Yaskawa INFORM job: aprem3TRJ0.JBI

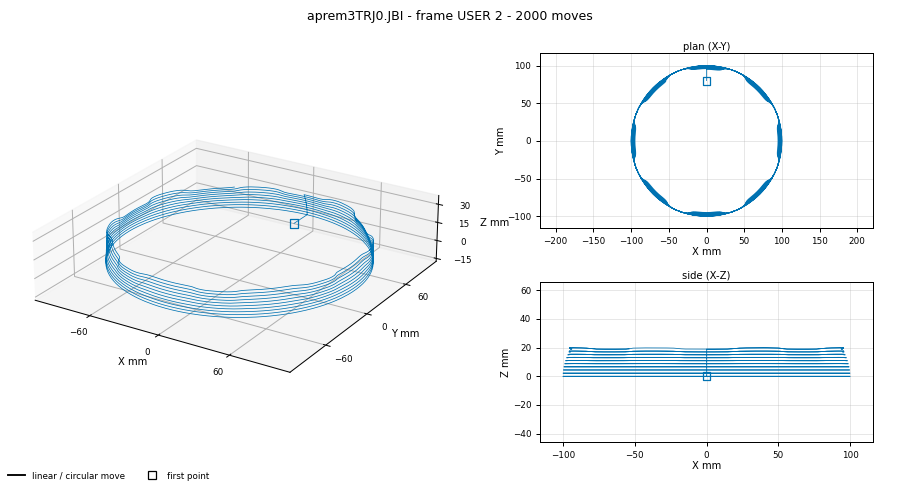
[picture p0: tool path of aprem3TRJ0.JBI in frame USER 2, 2000 of 2000 moves have a stored position in this frame; points joined in program order, loops and branches not executed]
/JOB
//NAME aprem3TRJ0
///FOLDERNAME DEMO
//POS
///NPOS 2000,0,2000,0,0,0
///USER 2
///TOOL 7
///POSTYPE USER
///RECTAN
///RCONF 1,0,0,0,0,0,0,0,0,0,0,0,0,0,0,0,0,0,0,0,0,0,0,0
C00000=0.000,80.000,0.000,-180.0000,0.0000,-0.0000
C00001=0.000,100.000,0.000,-180.0000,0.0000,-0.0000
C00002=5.792,99.832,0.000,-180.0000,-0.0000,-3.3204
C00003=10.988,99.394,0.000,-180.0000,-0.0000,-6.3084
C00004=15.564,98.781,0.000,-180.0000,-0.0000,-8.9540
C00005=18.698,98.237,0.000,-180.0000,-0.0000,-10.7765
C00006=20.854,97.801,0.000,-180.0000,-0.0000,-12.0369
C00007=22.593,97.414,0.000,-180.0000,-0.0000,-13.0576
C00008=24.351,96.990,0.000,-180.0000,-0.0000,-14.0938
C00009=26.550,96.411,0.000,-180.0000,-0.0000,-15.3967
C00010=29.248,95.627,0.000,-180.0000,-0.0000,-17.0065
C00011=32.094,94.710,0.000,-180.0000,-0.0000,-18.7198
C00012=34.739,93.772,0.000,-180.0000,-0.0000,-20.3278
C00013=37.121,92.855,0.000,-180.0000,-0.0000,-21.7902
C00014=39.410,91.907,0.000,-180.0000,-0.0000,-23.2098
C00015=41.743,90.871,0.000,-180.0000,-0.0000,-24.6724
C00016=44.276,89.664,0.000,180.0000,0.0000,-26.2801
C00017=46.937,88.300,0.000,180.0000,0.0000,-27.9935
C00018=49.400,86.946,0.000,-180.0000,-0.0000,-29.6039
C00019=51.363,85.801,0.000,-180.0000,-0.0000,-30.9060
C00020=52.906,84.858,0.000,-180.0000,-0.0000,-31.9421
C00021=54.410,83.902,0.000,-180.0000,-0.0000,-32.9632
C00022=56.242,82.685,0.000,-180.0000,-0.0000,-34.2234
C00023=58.844,80.854,0.000,-180.0000,-0.0000,-36.0464
C00024=62.512,78.053,0.000,-180.0000,-0.0000,-38.6909
C00025=66.496,74.687,0.000,-180.0000,-0.0000,-41.6796
C00026=70.711,70.711,0.000,-180.0000,-0.0000,-45.0000
C00027=74.687,66.496,0.000,-180.0000,-0.0000,-48.3204
C00028=78.053,62.512,0.000,-180.0000,-0.0000,-51.3091
C00029=80.854,58.844,0.000,180.0000,0.0000,-53.9536
C00030=82.685,56.242,0.000,-180.0000,-0.0000,-55.7766
C00031=83.902,54.410,0.000,-180.0000,-0.0000,-57.0368
C00032=84.858,52.906,0.000,-180.0000,-0.0000,-58.0579
C00033=85.801,51.363,0.000,-180.0000,-0.0000,-59.0940
C00034=86.946,49.400,0.000,-180.0000,-0.0000,-60.3961
C00035=88.300,46.937,0.000,-180.0000,-0.0000,-62.0065
C00036=89.664,44.276,0.000,-180.0000,-0.0000,-63.7199
C00037=90.871,41.743,0.000,-180.0000,-0.0000,-65.3276
C00038=91.907,39.410,0.000,-180.0000,-0.0000,-66.7902
C00039=92.855,37.121,0.000,-180.0000,-0.0000,-68.2098
C00040=93.772,34.739,0.000,-180.0000,-0.0000,-69.6722
C00041=94.710,32.094,0.000,-180.0000,-0.0000,-71.2802
C00042=95.627,29.248,0.000,-180.0000,-0.0000,-72.9935
C00043=96.411,26.550,0.000,-180.0000,-0.0000,-74.6033
C00044=96.990,24.351,0.000,-180.0000,-0.0000,-75.9062
C00045=97.414,22.593,0.000,-180.0000,-0.0000,-76.9424
C00046=97.801,20.854,0.000,-180.0000,-0.0000,-77.9631
C00047=98.237,18.698,0.000,-180.0000,-0.0000,-79.2235
C00048=98.781,15.564,0.000,-180.0000,-0.0000,-81.0460
C00049=99.394,10.988,0.000,-180.0000,-0.0000,-83.6916
C00050=99.832,5.792,0.000,-180.0000,-0.0000,-86.6796
C00051=100.000,0.000,0.000,-180.0000,-0.0000,-90.0000
C00052=99.832,-5.792,0.000,180.0000,-0.0000,-93.3204
C00053=99.394,-10.988,0.000,180.0000,-0.0000,-96.3084
C00054=98.781,-15.564,0.000,180.0000,-0.0000,-98.9540
C00055=98.237,-18.698,0.000,180.0000,-0.0000,-100.7765
C00056=97.801,-20.854,0.000,180.0000,-0.0000,-102.0369
C00057=97.414,-22.593,0.000,180.0000,-0.0000,-103.0576
C00058=96.990,-24.351,0.000,180.0000,-0.0000,-104.0938
C00059=96.411,-26.550,0.000,180.0000,-0.0000,-105.3967
C00060=95.627,-29.248,0.000,180.0000,-0.0000,-107.0065
C00061=94.710,-32.094,0.000,180.0000,-0.0000,-108.7198
C00062=93.772,-34.739,0.000,180.0000,-0.0000,-110.3278
C00063=92.855,-37.121,0.000,180.0000,-0.0000,-111.7902
C00064=91.907,-39.410,0.000,180.0000,-0.0000,-113.2098
C00065=90.871,-41.743,0.000,180.0000,-0.0000,-114.6724
C00066=89.664,-44.276,0.000,180.0000,-0.0000,-116.2801
C00067=88.300,-46.937,0.000,180.0000,-0.0000,-117.9935
C00068=86.946,-49.400,0.000,180.0000,-0.0000,-119.6039
C00069=85.801,-51.363,0.000,180.0000,-0.0000,-120.9060
C00070=84.858,-52.906,0.000,180.0000,-0.0000,-121.9421
C00071=83.902,-54.410,0.000,180.0000,-0.0000,-122.9632
C00072=82.685,-56.242,0.000,180.0000,-0.0000,-124.2234
C00073=80.854,-58.844,0.000,180.0000,-0.0000,-126.0464
C00074=78.053,-62.512,0.000,180.0000,-0.0000,-128.6909
C00075=74.687,-66.496,0.000,180.0000,-0.0000,-131.6796
C00076=70.711,-70.711,0.000,180.0000,-0.0000,-135.0000
C00077=66.496,-74.687,0.000,180.0000,-0.0000,-138.3204
C00078=62.512,-78.053,0.000,180.0000,-0.0000,-141.3091
C00079=58.844,-80.854,0.000,180.0000,-0.0000,-143.9536
C00080=56.242,-82.685,0.000,180.0000,-0.0000,-145.7766
C00081=54.410,-83.902,0.000,180.0000,-0.0000,-147.0368
C00082=52.906,-84.858,0.000,180.0000,-0.0000,-148.0579
C00083=51.363,-85.801,0.000,180.0000,-0.0000,-149.0940
C00084=49.400,-86.946,0.000,-180.0000,0.0000,-150.3961
C00085=46.937,-88.300,0.000,180.0000,-0.0000,-152.0065
C00086=44.276,-89.664,0.000,180.0000,-0.0000,-153.7199
C00087=41.743,-90.871,0.000,180.0000,-0.0000,-155.3276
C00088=39.410,-91.907,0.000,180.0000,-0.0000,-156.7902
C00089=37.121,-92.855,0.000,180.0000,-0.0000,-158.2098
C00090=34.739,-93.772,0.000,180.0000,-0.0000,-159.6722
C00091=32.094,-94.710,0.000,180.0000,-0.0000,-161.2802
C00092=29.248,-95.627,0.000,180.0000,-0.0000,-162.9935
C00093=26.550,-96.411,0.000,180.0000,-0.0000,-164.6033
C00094=24.351,-96.990,0.000,180.0000,-0.0000,-165.9062
C00095=22.593,-97.414,0.000,180.0000,-0.0000,-166.9424
C00096=20.854,-97.801,0.000,180.0000,-0.0000,-167.9631
C00097=18.698,-98.237,0.000,180.0000,-0.0000,-169.2235
C00098=15.564,-98.781,0.000,180.0000,-0.0000,-171.0460
C00099=10.988,-99.394,0.000,180.0000,-0.0000,-173.6916
C00100=5.792,-99.832,0.000,180.0000,-0.0000,-176.6796
C00101=0.000,-100.000,0.000,-180.0000,-0.0000,-180.0000
C00102=0.000,-100.000,0.000,-180.0000,-0.0000,-180.0000
C00103=-5.792,-99.832,0.000,-180.0000,-0.0000,-183.3204
C00104=-10.988,-99.394,0.000,-180.0000,-0.0000,-186.3084
C00105=-15.564,-98.781,0.000,-180.0000,-0.0000,-188.9540
C00106=-18.698,-98.237,0.000,-180.0000,-0.0000,-190.7765
C00107=-20.854,-97.801,0.000,-180.0000,-0.0000,-192.0369
C00108=-22.593,-97.414,0.000,-180.0000,-0.0000,-193.0576
C00109=-24.351,-96.990,0.000,-180.0000,-0.0000,-194.0938
C00110=-26.550,-96.411,0.000,-180.0000,-0.0000,-195.3967
C00111=-29.248,-95.627,0.000,-180.0000,-0.0000,-197.0065
C00112=-32.094,-94.710,0.000,-180.0000,-0.0000,-198.7198
C00113=-34.739,-93.772,0.000,-180.0000,-0.0000,-200.3278
C00114=-37.121,-92.855,0.000,-180.0000,-0.0000,-201.7902
C00115=-39.410,-91.907,0.000,-180.0000,-0.0000,-203.2098
C00116=-41.743,-90.871,0.000,-180.0000,-0.0000,-204.6724
C00117=-44.276,-89.664,0.000,-180.0000,-0.0000,-206.2801
C00118=-46.937,-88.300,0.000,-180.0000,-0.0000,-207.9935
C00119=-49.400,-86.946,0.000,-180.0000,-0.0000,-209.6039
C00120=-51.363,-85.801,0.000,-180.0000,-0.0000,-210.9060
C00121=-52.906,-84.858,0.000,-180.0000,-0.0000,-211.9421
C00122=-54.410,-83.902,0.000,-180.0000,-0.0000,-212.9632
C00123=-56.242,-82.685,0.000,-180.0000,-0.0000,-214.2234
C00124=-58.844,-80.854,0.000,-180.0000,-0.0000,-216.0464
C00125=-62.512,-78.053,0.000,-180.0000,-0.0000,-218.6909
C00126=-66.496,-74.687,0.000,-180.0000,-0.0000,-221.6796
C00127=-70.711,-70.711,0.000,-180.0000,-0.0000,-225.0000
C00128=-74.687,-66.496,0.000,-180.0000,-0.0000,-228.3204
C00129=-78.053,-62.512,0.000,-180.0000,-0.0000,-231.3091
C00130=-80.854,-58.844,0.000,-180.0000,-0.0000,-233.9536
C00131=-82.685,-56.242,0.000,-180.0000,-0.0000,-235.7766
C00132=-83.902,-54.410,0.000,-180.0000,-0.0000,-237.0368
C00133=-84.858,-52.906,0.000,-180.0000,-0.0000,-238.0579
C00134=-85.801,-51.363,0.000,-180.0000,-0.0000,-239.0940
C00135=-86.946,-49.400,0.000,-180.0000,-0.0000,-240.3961
C00136=-88.300,-46.937,0.000,-180.0000,-0.0000,-242.0065
C00137=-89.664,-44.276,0.000,-180.0000,-0.0000,-243.7199
C00138=-90.871,-41.743,0.000,180.0000,0.0000,-245.3276
C00139=-91.907,-39.410,0.000,180.0000,0.0000,-246.7902
C00140=-92.855,-37.121,0.000,-180.0000,-0.0000,-248.2098
C00141=-93.772,-34.739,0.000,-180.0000,-0.0000,-249.6722
C00142=-94.710,-32.094,0.000,180.0000,0.0000,-251.2802
C00143=-95.627,-29.248,0.000,180.0000,0.0000,-252.9935
C00144=-96.411,-26.550,0.000,-180.0000,-0.0000,-254.6033
C00145=-96.990,-24.351,0.000,-180.0000,-0.0000,-255.9062
C00146=-97.414,-22.593,0.000,-180.0000,-0.0000,-256.9424
C00147=-97.801,-20.854,0.000,-180.0000,-0.0000,-257.9631
C00148=-98.237,-18.698,0.000,-180.0000,-0.0000,-259.2235
C00149=-98.781,-15.564,0.000,-180.0000,-0.0000,-261.0460
C00150=-99.394,-10.988,0.000,-180.0000,-0.0000,-263.6916
C00151=-99.832,-5.792,0.000,-180.0000,-0.0000,-266.6796
C00152=-100.000,0.000,0.000,180.0000,0.0000,-270.0000
C00153=-99.832,5.792,0.000,-180.0000,0.0000,-273.3204
C00154=-99.394,10.988,0.000,-180.0000,0.0000,-276.3084
C00155=-98.781,15.564,0.000,-180.0000,0.0000,-278.9540
C00156=-98.237,18.698,0.000,-180.0000,0.0000,-280.7765
C00157=-97.801,20.854,0.000,-180.0000,0.0000,-282.0369
C00158=-97.414,22.593,0.000,-180.0000,0.0000,-283.0576
C00159=-96.990,24.351,0.000,-180.0000,0.0000,-284.0938
C00160=-96.411,26.550,0.000,-180.0000,0.0000,-285.3967
C00161=-95.627,29.248,0.000,-180.0000,0.0000,-287.0065
C00162=-94.710,32.094,0.000,-180.0000,0.0000,-288.7198
C00163=-93.772,34.739,0.000,-180.0000,0.0000,-290.3278
C00164=-92.855,37.121,0.000,-180.0000,0.0000,-291.7902
C00165=-91.907,39.410,0.000,-180.0000,0.0000,-293.2098
C00166=-90.871,41.743,0.000,-180.0000,0.0000,-294.6724
C00167=-89.664,44.276,0.000,-180.0000,0.0000,-296.2801
C00168=-88.300,46.937,0.000,-180.0000,0.0000,-297.9935
C00169=-86.946,49.400,0.000,-180.0000,0.0000,-299.6039
C00170=-85.801,51.363,0.000,-180.0000,0.0000,-300.9060
C00171=-84.858,52.906,0.000,-180.0000,0.0000,-301.9421
C00172=-83.902,54.410,0.000,-180.0000,0.0000,-302.9632
C00173=-82.685,56.242,0.000,-180.0000,0.0000,-304.2234
C00174=-80.854,58.844,0.000,-180.0000,0.0000,-306.0464
C00175=-78.053,62.512,0.000,-180.0000,0.0000,-308.6909
C00176=-74.687,66.496,0.000,-180.0000,0.0000,-311.6796
C00177=-70.711,70.711,0.000,-180.0000,0.0000,-315.0000
C00178=-66.496,74.687,0.000,-180.0000,0.0000,-318.3204
C00179=-62.512,78.053,0.000,-180.0000,0.0000,-321.3091
C00180=-58.844,80.854,0.000,-180.0000,0.0000,-323.9536
C00181=-56.242,82.685,0.000,-180.0000,0.0000,-325.7766
C00182=-54.410,83.902,0.000,-180.0000,0.0000,-327.0368
C00183=-52.906,84.858,0.000,-180.0000,0.0000,-328.0579
C00184=-51.363,85.801,0.000,-180.0000,0.0000,-329.0940
C00185=-49.400,86.946,0.000,-180.0000,0.0000,-330.3961
C00186=-46.937,88.300,0.000,-180.0000,0.0000,-332.0065
C00187=-44.276,89.664,0.000,-180.0000,0.0000,-333.7199
C00188=-41.743,90.871,0.000,-180.0000,0.0000,-335.3276
C00189=-39.410,91.907,0.000,-180.0000,0.0000,-336.7902
C00190=-37.121,92.855,0.000,-180.0000,0.0000,-338.2098
C00191=-34.739,93.772,0.000,-180.0000,0.0000,-339.6722
C00192=-32.094,94.710,0.000,-180.0000,0.0000,-341.2802
C00193=-29.248,95.627,0.000,-180.0000,0.0000,-342.9935
C00194=-26.550,96.411,0.000,-180.0000,0.0000,-344.6033
C00195=-24.351,96.990,0.000,-180.0000,0.0000,-345.9062
C00196=-22.593,97.414,0.000,-180.0000,0.0000,-346.9424
C00197=-20.854,97.801,0.000,-180.0000,0.0000,-347.9631
C00198=-18.698,98.237,0.000,-180.0000,0.0000,-349.2235
C00199=-15.564,98.781,0.000,-180.0000,0.0000,-351.0460
C00200=-10.988,99.394,0.000,-180.0000,0.0000,-353.6916
C00201=-5.792,99.832,0.000,-180.0000,0.0000,-356.6796
C00202=0.000,100.000,0.000,-180.0000,0.0000,-360.0000
C00203=0.000,99.921,2.199,-175.9398,0.0000,-360.0000
C00204=5.785,99.754,2.199,-175.9444,-0.2364,-363.3190
C00205=10.976,99.317,2.199,-175.9703,-0.4452,-366.3064
C00206=15.549,98.707,2.199,-176.1463,-0.6026,-368.9521
C00207=18.681,98.171,2.199,-176.5600,-0.6415,-370.7740
C00208=20.835,97.748,2.199,-177.1484,-0.5884,-372.0325
C00209=22.573,97.375,2.200,-177.8314,-0.4845,-373.0515
C00210=24.330,96.965,2.200,-178.5159,-0.3619,-374.0856
C00211=26.527,96.399,2.200,-179.1045,-0.2425,-375.3858
C00212=29.226,95.625,2.200,-179.5721,-0.1295,-376.9948
C00213=32.077,94.713,2.200,-179.8787,-0.0409,-378.7100
C00214=34.728,93.776,2.200,-179.9807,-0.0071,-380.3211
C00215=37.118,92.856,2.200,-179.9977,-0.0009,-381.7884
C00216=39.413,91.905,2.200,-179.9978,-0.0010,-383.2118
C00217=41.753,90.866,2.200,-179.9813,-0.0086,-384.6788
C00218=44.291,89.654,2.200,-179.8853,-0.0569,-386.2904
C00219=46.951,88.283,2.200,-179.6059,-0.2110,-388.0051
C00220=49.407,86.922,2.200,-179.1953,-0.4618,-389.6142
C00221=51.360,85.768,2.200,-178.6947,-0.7937,-390.9142
C00222=52.893,84.816,2.200,-178.1239,-1.1914,-391.9485
C00223=54.385,83.851,2.199,-177.5673,-1.6016,-392.9671
C00224=56.208,82.627,2.199,-177.1135,-1.9809,-394.2260
C00225=58.802,80.791,2.199,-176.8480,-2.3017,-396.0482
C00226=62.466,77.989,2.199,-176.8343,-2.5377,-398.6933
C00227=66.446,74.627,2.199,-176.9631,-2.7034,-401.6811
C00228=70.655,70.655,2.199,-177.1266,-2.8734,-405.0000
C00229=74.627,66.446,2.199,-177.2966,-3.0369,-408.3189
C00230=77.989,62.466,2.199,-177.4623,-3.1657,-411.3067
C00231=80.791,58.802,2.199,-177.6983,-3.1520,-413.9518
C00232=82.627,56.208,2.199,-178.0191,-2.8865,-415.7740
C00233=83.851,54.385,2.199,-178.3984,-2.4327,-417.0329
C00234=84.816,52.893,2.200,-178.8086,-1.8761,-418.0515
C00235=85.768,51.360,2.200,-179.2063,-1.3053,-419.0858
C00236=86.922,49.407,2.200,-179.5382,-0.8047,-420.3858
C00237=88.283,46.951,2.200,-179.7890,-0.3941,-421.9949
C00238=89.654,44.291,2.200,-179.9431,-0.1147,-423.7096
C00239=90.866,41.753,2.200,-179.9914,-0.0187,-425.3212
C00240=91.905,39.413,2.200,-179.9990,-0.0022,-426.7882
C00241=92.856,37.118,2.200,-179.9991,-0.0023,-428.2116
C00242=93.776,34.728,2.200,-179.9929,-0.0193,-429.6789
C00243=94.713,32.077,2.200,-179.9591,-0.1213,-431.2900
C00244=95.625,29.226,2.200,-179.8705,-0.4279,-433.0052
C00245=96.399,26.527,2.200,-179.7575,-0.8955,-434.6142
C00246=96.965,24.330,2.200,-179.6381,-1.4841,-435.9144
C00247=97.375,22.573,2.200,-179.5155,-2.1686,-436.9485
C00248=97.748,20.835,2.199,-179.4116,-2.8516,-437.9675
C00249=98.171,18.681,2.199,-179.3585,-3.4400,-439.2260
C00250=98.707,15.549,2.199,-179.3974,-3.8537,-441.0479
C00251=99.317,10.976,2.199,-179.5548,-4.0297,-443.6936
C00252=99.754,5.785,2.199,-179.7636,-4.0556,-446.6810
C00253=99.921,0.000,2.199,180.0000,-4.0602,-450.0000
C00254=99.754,-5.785,2.199,179.7636,-4.0556,-453.3190
C00255=99.317,-10.976,2.199,179.5548,-4.0297,-456.3064
C00256=98.707,-15.549,2.199,179.3974,-3.8537,-458.9521
C00257=98.171,-18.681,2.199,179.3585,-3.4400,-460.7740
C00258=97.748,-20.835,2.199,179.4116,-2.8516,-462.0325
C00259=97.375,-22.573,2.200,179.5155,-2.1686,-463.0515
C00260=96.965,-24.330,2.200,179.6381,-1.4841,-464.0856
C00261=96.399,-26.527,2.200,179.7575,-0.8955,-465.3858
C00262=95.625,-29.226,2.200,179.8705,-0.4279,-466.9948
C00263=94.713,-32.077,2.200,179.9591,-0.1213,-468.7100
C00264=93.776,-34.728,2.200,179.9929,-0.0193,-470.3211
C00265=92.856,-37.118,2.200,179.9991,-0.0023,-471.7884
C00266=91.905,-39.413,2.200,179.9990,-0.0022,-473.2118
C00267=90.866,-41.753,2.200,179.9914,-0.0187,-474.6788
C00268=89.654,-44.291,2.200,179.9431,-0.1147,-476.2904
C00269=88.283,-46.951,2.200,179.7890,-0.3941,-478.0051
C00270=86.922,-49.407,2.200,179.5382,-0.8047,-479.6142
C00271=85.768,-51.360,2.200,179.2063,-1.3053,-480.9142
C00272=84.816,-52.893,2.200,178.8086,-1.8761,-481.9485
C00273=83.851,-54.385,2.199,178.3984,-2.4327,-482.9671
C00274=82.627,-56.208,2.199,178.0191,-2.8865,-484.2260
C00275=80.791,-58.802,2.199,177.6983,-3.1520,-486.0482
C00276=77.989,-62.466,2.199,177.4623,-3.1657,-488.6933
C00277=74.627,-66.446,2.199,177.2966,-3.0369,-491.6811
C00278=70.655,-70.655,2.199,177.1266,-2.8734,-495.0000
C00279=66.446,-74.627,2.199,176.9631,-2.7034,-498.3189
C00280=62.466,-77.989,2.199,176.8343,-2.5377,-501.3067
C00281=58.802,-80.791,2.199,176.8480,-2.3017,-503.9518
C00282=56.208,-82.627,2.199,177.1135,-1.9809,-505.7740
C00283=54.385,-83.851,2.199,177.5673,-1.6016,-507.0329
C00284=52.893,-84.816,2.200,178.1239,-1.1914,-508.0515
C00285=51.360,-85.768,2.200,178.6947,-0.7937,-509.0858
C00286=49.407,-86.922,2.200,179.1953,-0.4618,-510.3858
C00287=46.951,-88.283,2.200,179.6059,-0.2110,-511.9949
C00288=44.291,-89.654,2.200,179.8853,-0.0569,-513.7096
C00289=41.753,-90.866,2.200,179.9813,-0.0086,-515.3212
C00290=39.413,-91.905,2.200,179.9978,-0.0010,-516.7882
C00291=37.118,-92.856,2.200,179.9977,-0.0009,-518.2116
C00292=34.728,-93.776,2.200,179.9807,-0.0071,-519.6789
C00293=32.077,-94.713,2.200,179.8787,-0.0409,-521.2900
C00294=29.226,-95.625,2.200,179.5721,-0.1295,-523.0052
C00295=26.527,-96.399,2.200,179.1045,-0.2425,-524.6142
C00296=24.330,-96.965,2.200,178.5159,-0.3619,-525.9144
C00297=22.573,-97.375,2.200,177.8314,-0.4845,-526.9485
C00298=20.835,-97.748,2.199,177.1484,-0.5884,-527.9675
C00299=18.681,-98.171,2.199,176.5600,-0.6415,-529.2260
C00300=15.549,-98.707,2.199,176.1463,-0.6026,-531.0479
C00301=10.976,-99.317,2.199,175.9703,-0.4452,-533.6936
C00302=5.785,-99.754,2.199,175.9444,-0.2364,-536.6810
C00303=0.000,-99.921,2.199,175.9398,0.0000,-540.0000
C00304=0.000,-99.921,2.199,175.9398,0.0000,-540.0000
C00305=-5.785,-99.754,2.199,175.9444,0.2364,-543.3190
C00306=-10.976,-99.317,2.199,175.9703,0.4452,-546.3064
C00307=-15.549,-98.707,2.199,176.1463,0.6026,-548.9521
C00308=-18.681,-98.171,2.199,176.5600,0.6415,-550.7740
C00309=-20.835,-97.748,2.199,177.1484,0.5884,-552.0325
C00310=-22.573,-97.375,2.200,177.8314,0.4845,-553.0515
C00311=-24.330,-96.965,2.200,178.5159,0.3619,-554.0856
C00312=-26.527,-96.399,2.200,179.1045,0.2425,-555.3858
C00313=-29.226,-95.625,2.200,179.5721,0.1295,-556.9948
C00314=-32.077,-94.713,2.200,179.8787,0.0409,-558.7100
C00315=-34.728,-93.776,2.200,179.9807,0.0071,-560.3211
C00316=-37.118,-92.856,2.200,179.9977,0.0009,-561.7884
C00317=-39.413,-91.905,2.200,179.9978,0.0010,-563.2118
C00318=-41.753,-90.866,2.200,179.9813,0.0086,-564.6788
C00319=-44.291,-89.654,2.200,179.8853,0.0569,-566.2904
C00320=-46.951,-88.283,2.200,179.6059,0.2110,-568.0051
C00321=-49.407,-86.922,2.200,179.1953,0.4618,-569.6142
C00322=-51.360,-85.768,2.200,178.6947,0.7937,-570.9142
C00323=-52.893,-84.816,2.200,178.1239,1.1914,-571.9485
C00324=-54.385,-83.851,2.199,177.5673,1.6016,-572.9671
C00325=-56.208,-82.627,2.199,177.1135,1.9809,-574.2260
C00326=-58.802,-80.791,2.199,176.8480,2.3017,-576.0482
C00327=-62.466,-77.989,2.199,176.8343,2.5377,-578.6933
C00328=-66.446,-74.627,2.199,176.9631,2.7034,-581.6811
C00329=-70.655,-70.655,2.199,177.1266,2.8734,-585.0000
C00330=-74.627,-66.446,2.199,177.2966,3.0369,-588.3189
C00331=-77.989,-62.466,2.199,177.4623,3.1657,-591.3067
C00332=-80.791,-58.802,2.199,177.6983,3.1520,-593.9518
C00333=-82.627,-56.208,2.199,178.0191,2.8865,-595.7740
C00334=-83.851,-54.385,2.199,178.3984,2.4327,-597.0329
C00335=-84.816,-52.893,2.200,178.8086,1.8761,-598.0515
C00336=-85.768,-51.360,2.200,179.2063,1.3053,-599.0858
C00337=-86.922,-49.407,2.200,179.5382,0.8047,-600.3858
C00338=-88.283,-46.951,2.200,179.7890,0.3941,-601.9949
C00339=-89.654,-44.291,2.200,179.9431,0.1147,-603.7096
C00340=-90.866,-41.753,2.200,179.9914,0.0187,-605.3212
C00341=-91.905,-39.413,2.200,179.9990,0.0022,-606.7882
C00342=-92.856,-37.118,2.200,179.9991,0.0023,-608.2116
C00343=-93.776,-34.728,2.200,179.9929,0.0193,-609.6789
C00344=-94.713,-32.077,2.200,179.9591,0.1213,-611.2900
C00345=-95.625,-29.226,2.200,179.8705,0.4279,-613.0052
C00346=-96.399,-26.527,2.200,179.7575,0.8955,-614.6142
C00347=-96.965,-24.330,2.200,179.6381,1.4841,-615.9144
C00348=-97.375,-22.573,2.200,179.5155,2.1686,-616.9485
C00349=-97.748,-20.835,2.199,179.4116,2.8516,-617.9675
C00350=-98.171,-18.681,2.199,179.3585,3.4400,-619.2260
C00351=-98.707,-15.549,2.199,179.3974,3.8537,-621.0479
C00352=-99.317,-10.976,2.199,179.5548,4.0297,-623.6936
C00353=-99.754,-5.785,2.199,179.7636,4.0556,-626.6810
C00354=-99.921,0.000,2.199,-180.0000,4.0602,-630.0000
C00355=-99.754,5.785,2.199,-179.7636,4.0556,-633.3190
C00356=-99.317,10.976,2.199,-179.5548,4.0297,-636.3064
C00357=-98.707,15.549,2.199,-179.3974,3.8537,-638.9521
C00358=-98.171,18.681,2.199,-179.3585,3.4400,-640.7740
C00359=-97.748,20.835,2.199,-179.4116,2.8516,-642.0325
C00360=-97.375,22.573,2.200,-179.5155,2.1686,-643.0515
C00361=-96.965,24.330,2.200,-179.6381,1.4841,-644.0856
C00362=-96.399,26.527,2.200,-179.7575,0.8955,-645.3858
C00363=-95.625,29.226,2.200,-179.8705,0.4279,-646.9948
C00364=-94.713,32.077,2.200,-179.9591,0.1213,-648.7100
C00365=-93.776,34.728,2.200,-179.9929,0.0193,-650.3211
C00366=-92.856,37.118,2.200,-179.9991,0.0023,-651.7884
C00367=-91.905,39.413,2.200,-179.9990,0.0022,-653.2118
C00368=-90.866,41.753,2.200,-179.9914,0.0187,-654.6788
C00369=-89.654,44.291,2.200,-179.9431,0.1147,-656.2904
C00370=-88.283,46.951,2.200,-179.7890,0.3941,-658.0051
C00371=-86.922,49.407,2.200,-179.5382,0.8047,-659.6142
C00372=-85.768,51.360,2.200,-179.2063,1.3053,-660.9142
C00373=-84.816,52.893,2.200,-178.8086,1.8761,-661.9485
C00374=-83.851,54.385,2.199,-178.3984,2.4327,-662.9671
C00375=-82.627,56.208,2.199,-178.0191,2.8865,-664.2260
C00376=-80.791,58.802,2.199,-177.6983,3.1520,-666.0482
C00377=-77.989,62.466,2.199,-177.4623,3.1657,-668.6933
C00378=-74.627,66.446,2.199,-177.2966,3.0369,-671.6811
C00379=-70.655,70.655,2.199,-177.1266,2.8734,-675.0000
C00380=-66.446,74.627,2.199,-176.9631,2.7034,-678.3189
C00381=-62.466,77.989,2.199,-176.8343,2.5377,-681.3067
C00382=-58.802,80.791,2.199,-176.8480,2.3017,-683.9518
C00383=-56.208,82.627,2.199,-177.1135,1.9809,-685.7740
C00384=-54.385,83.851,2.199,-177.5673,1.6016,-687.0329
C00385=-52.893,84.816,2.200,-178.1239,1.1914,-688.0515
C00386=-51.360,85.768,2.200,-178.6947,0.7937,-689.0858
C00387=-49.407,86.922,2.200,-179.1953,0.4618,-690.3858
C00388=-46.951,88.283,2.200,-179.6059,0.2110,-691.9949
C00389=-44.291,89.654,2.200,-179.8853,0.0569,-693.7096
C00390=-41.753,90.866,2.200,-179.9813,0.0086,-695.3212
C00391=-39.413,91.905,2.200,-179.9978,0.0010,-696.7882
C00392=-37.118,92.856,2.200,-179.9977,0.0009,-698.2116
C00393=-34.728,93.776,2.200,-179.9807,0.0071,-699.6789
C00394=-32.077,94.713,2.200,-179.8787,0.0409,-701.2900
C00395=-29.226,95.625,2.200,-179.5721,0.1295,-703.0052
C00396=-26.527,96.399,2.200,-179.1045,0.2425,-704.6142
C00397=-24.330,96.965,2.200,-178.5159,0.3619,-705.9144
C00398=-22.573,97.375,2.200,-177.8314,0.4845,-706.9485
C00399=-20.835,97.748,2.199,-177.1484,0.5884,-707.9675
C00400=-18.681,98.171,2.199,-176.5600,0.6415,-709.2260
C00401=-15.549,98.707,2.199,-176.1463,0.6026,-711.0479
C00402=-10.976,99.317,2.199,-175.9703,0.4452,-713.6936
C00403=-5.785,99.754,2.199,-175.9444,0.2364,-716.6810
C00404=0.000,99.921,2.199,-175.9398,0.0000,-720.0000
C00405=0.000,99.691,4.387,-172.1026,0.0000,-720.0000
C00406=5.764,99.524,4.387,-172.1115,-0.4617,-723.3146
C00407=10.941,99.090,4.387,-172.1612,-0.8645,-726.3008
C00408=15.506,98.490,4.388,-172.4978,-1.1464,-728.9471
C00409=18.630,97.979,4.390,-173.2935,-1.1748,-730.7659
C00410=20.779,97.591,4.393,-174.4370,-1.0358,-732.0199
C00411=22.514,97.259,4.396,-175.7755,-0.8390,-733.0335
C00412=24.268,96.890,4.398,-177.1185,-0.6429,-734.0616
C00413=26.460,96.362,4.399,-178.2686,-0.4458,-735.3544
C00414=29.164,95.617,4.399,-179.1783,-0.2412,-736.9622
C00415=32.027,94.722,4.399,-179.7705,-0.0761,-738.6812
C00416=34.697,93.786,4.400,-179.9632,-0.0136,-740.3024
C00417=37.107,92.860,4.400,-179.9957,-0.0017,-741.7817
C00418=39.424,91.901,4.400,-179.9957,-0.0018,-743.2185
C00419=41.782,90.851,4.400,-179.9644,-0.0164,-744.6975
C00420=44.332,89.625,4.399,-179.7839,-0.1085,-746.3188
C00421=46.990,88.233,4.399,-179.2484,-0.4105,-748.0383
C00422=49.428,86.848,4.399,-178.4605,-0.9093,-749.6456
C00423=51.352,85.672,4.398,-177.5077,-1.5842,-750.9386
C00424=52.853,84.692,4.396,-176.4188,-2.3979,-751.9667
C00425=54.314,83.700,4.393,-175.3318,-3.2102,-752.9801
C00426=56.108,82.455,4.390,-174.4229,-3.9270,-754.2340
C00427=58.679,80.608,4.388,-173.8773,-4.5153,-756.0529
C00428=62.331,77.804,4.387,-173.8348,-4.9540,-758.6992
C00429=66.299,74.450,4.387,-174.0811,-5.2722,-761.6856
C00430=70.493,70.493,4.387,-174.3980,-5.6020,-765.0000
C00431=74.450,66.299,4.387,-174.7278,-5.9188,-768.3144
C00432=77.804,62.331,4.387,-175.0460,-6.1652,-771.3008
C00433=80.608,58.679,4.388,-175.4847,-6.1227,-773.9471
C00434=82.455,56.108,4.390,-176.0730,-5.5771,-775.7660
C00435=83.700,54.314,4.393,-176.7898,-4.6682,-777.0199
C00436=84.692,52.853,4.396,-177.6021,-3.5812,-778.0333
C00437=85.672,51.352,4.398,-178.4158,-2.4923,-779.0614
C00438=86.848,49.428,4.399,-179.0907,-1.5395,-780.3544
C00439=88.233,46.990,4.399,-179.5895,-0.7516,-781.9617
C00440=89.625,44.332,4.399,-179.8915,-0.2161,-783.6812
C00441=90.851,41.782,4.400,-179.9836,-0.0356,-785.3025
C00442=91.901,39.424,4.400,-179.9982,-0.0043,-786.7815
C00443=92.860,37.107,4.400,-179.9983,-0.0043,-788.2183
C00444=93.786,34.697,4.400,-179.9864,-0.0368,-789.6976
C00445=94.722,32.027,4.399,-179.9239,-0.2295,-791.3188
C00446=95.617,29.164,4.399,-179.7588,-0.8217,-793.0378
C00447=96.362,26.460,4.399,-179.5542,-1.7314,-794.6456
C00448=96.890,24.268,4.398,-179.3571,-2.8815,-795.9384
C00449=97.259,22.514,4.396,-179.1610,-4.2245,-796.9665
C00450=97.591,20.779,4.393,-178.9642,-5.5630,-797.9801
C00451=97.979,18.630,4.390,-178.8252,-6.7065,-799.2341
C00452=98.490,15.506,4.388,-178.8536,-7.5022,-801.0529
C00453=99.090,10.941,4.387,-179.1355,-7.8388,-803.6992
C00454=99.524,5.764,4.387,-179.5383,-7.8885,-806.6854
C00455=99.691,0.000,4.387,180.0000,-7.8974,-810.0000
C00456=99.524,-5.764,4.387,179.5383,-7.8885,-813.3146
C00457=99.090,-10.941,4.387,179.1355,-7.8388,-816.3008
C00458=98.490,-15.506,4.388,178.8536,-7.5022,-818.9471
C00459=97.979,-18.630,4.390,178.8252,-6.7065,-820.7659
C00460=97.591,-20.779,4.393,178.9642,-5.5630,-822.0199
C00461=97.259,-22.514,4.396,179.1610,-4.2245,-823.0335
C00462=96.890,-24.268,4.398,179.3571,-2.8815,-824.0616
C00463=96.362,-26.460,4.399,179.5542,-1.7314,-825.3544
C00464=95.617,-29.164,4.399,179.7588,-0.8217,-826.9622
C00465=94.722,-32.027,4.399,179.9239,-0.2295,-828.6812
C00466=93.786,-34.697,4.400,179.9864,-0.0368,-830.3024
C00467=92.860,-37.107,4.400,179.9983,-0.0043,-831.7817
C00468=91.901,-39.424,4.400,179.9982,-0.0043,-833.2185
C00469=90.851,-41.782,4.400,179.9836,-0.0356,-834.6975
C00470=89.625,-44.332,4.399,179.8915,-0.2161,-836.3188
C00471=88.233,-46.990,4.399,179.5895,-0.7516,-838.0383
C00472=86.848,-49.428,4.399,179.0907,-1.5395,-839.6456
C00473=85.672,-51.352,4.398,178.4158,-2.4923,-840.9386
C00474=84.692,-52.853,4.396,177.6021,-3.5812,-841.9667
C00475=83.700,-54.314,4.393,176.7898,-4.6682,-842.9801
C00476=82.455,-56.108,4.390,176.0730,-5.5771,-844.2340
C00477=80.608,-58.679,4.388,175.4847,-6.1227,-846.0529
C00478=77.804,-62.331,4.387,175.0460,-6.1652,-848.6992
C00479=74.450,-66.299,4.387,174.7278,-5.9189,-851.6856
C00480=70.493,-70.493,4.387,174.3980,-5.6020,-855.0000
C00481=66.299,-74.450,4.387,174.0812,-5.2722,-858.3144
C00482=62.331,-77.804,4.387,173.8348,-4.9540,-861.3008
C00483=58.679,-80.608,4.388,173.8773,-4.5153,-863.9471
C00484=56.108,-82.455,4.390,174.4229,-3.9270,-865.7660
C00485=54.314,-83.700,4.393,175.3318,-3.2102,-867.0199
C00486=52.853,-84.692,4.396,176.4188,-2.3979,-868.0333
C00487=51.352,-85.672,4.398,177.5077,-1.5842,-869.0614
C00488=49.428,-86.848,4.399,178.4605,-0.9093,-870.3544
C00489=46.990,-88.233,4.399,179.2484,-0.4105,-871.9617
C00490=44.332,-89.625,4.399,179.7839,-0.1085,-873.6812
C00491=41.782,-90.851,4.400,179.9644,-0.0164,-875.3025
C00492=39.424,-91.901,4.400,179.9957,-0.0018,-876.7815
C00493=37.107,-92.860,4.400,179.9957,-0.0017,-878.2183
C00494=34.697,-93.786,4.400,179.9632,-0.0136,-879.6976
C00495=32.027,-94.722,4.399,179.7705,-0.0761,-881.3188
C00496=29.164,-95.617,4.399,179.1783,-0.2412,-883.0378
C00497=26.460,-96.362,4.399,178.2686,-0.4458,-884.6456
C00498=24.268,-96.890,4.398,177.1185,-0.6429,-885.9384
C00499=22.514,-97.259,4.396,175.7755,-0.8390,-886.9665
C00500=20.779,-97.591,4.393,174.4370,-1.0358,-887.9801
C00501=18.630,-97.979,4.390,173.2935,-1.1748,-889.2341
C00502=15.506,-98.490,4.388,172.4978,-1.1464,-891.0529
C00503=10.941,-99.090,4.387,172.1612,-0.8645,-893.6992
C00504=5.764,-99.524,4.387,172.1115,-0.4617,-896.6854
C00505=0.000,-99.691,4.387,172.1026,0.0000,-900.0000
C00506=0.000,-99.691,4.387,172.1026,0.0000,-900.0000
C00507=-5.764,-99.524,4.387,172.1115,0.4617,-903.3146
C00508=-10.941,-99.090,4.387,172.1612,0.8645,-906.3008
C00509=-15.506,-98.490,4.388,172.4978,1.1464,-908.9471
C00510=-18.630,-97.979,4.390,173.2935,1.1748,-910.7659
C00511=-20.779,-97.591,4.393,174.4370,1.0358,-912.0199
C00512=-22.514,-97.259,4.396,175.7755,0.8390,-913.0335
C00513=-24.268,-96.890,4.398,177.1185,0.6429,-914.0616
C00514=-26.460,-96.362,4.399,178.2686,0.4458,-915.3544
C00515=-29.164,-95.617,4.399,179.1783,0.2412,-916.9622
C00516=-32.027,-94.722,4.399,179.7705,0.0761,-918.6812
C00517=-34.697,-93.786,4.400,179.9632,0.0136,-920.3024
C00518=-37.107,-92.860,4.400,179.9957,0.0017,-921.7817
C00519=-39.424,-91.901,4.400,179.9957,0.0018,-923.2185
C00520=-41.782,-90.851,4.400,179.9644,0.0164,-924.6975
C00521=-44.332,-89.625,4.399,179.7839,0.1085,-926.3188
C00522=-46.990,-88.233,4.399,179.2484,0.4105,-928.0383
C00523=-49.428,-86.848,4.399,178.4605,0.9093,-929.6456
C00524=-51.352,-85.672,4.398,177.5077,1.5842,-930.9386
C00525=-52.853,-84.692,4.396,176.4188,2.3979,-931.9667
C00526=-54.314,-83.700,4.393,175.3318,3.2102,-932.9801
C00527=-56.108,-82.455,4.390,174.4229,3.9270,-934.2340
C00528=-58.679,-80.608,4.388,173.8773,4.5153,-936.0529
C00529=-62.331,-77.804,4.387,173.8348,4.9540,-938.6992
C00530=-66.299,-74.450,4.387,174.0811,5.2722,-941.6856
C00531=-70.493,-70.493,4.387,174.3980,5.6020,-945.0000
C00532=-74.450,-66.299,4.387,174.7278,5.9188,-948.3144
C00533=-77.804,-62.331,4.387,175.0460,6.1652,-951.3008
C00534=-80.608,-58.679,4.388,175.4847,6.1227,-953.9471
C00535=-82.455,-56.108,4.390,176.0730,5.5771,-955.7660
C00536=-83.700,-54.314,4.393,176.7898,4.6682,-957.0199
C00537=-84.692,-52.853,4.396,177.6021,3.5812,-958.0333
C00538=-85.672,-51.352,4.398,178.4158,2.4923,-959.0614
C00539=-86.848,-49.428,4.399,179.0907,1.5395,-960.3544
C00540=-88.233,-46.990,4.399,179.5895,0.7516,-961.9617
C00541=-89.625,-44.332,4.399,179.8915,0.2161,-963.6812
C00542=-90.851,-41.782,4.400,179.9836,0.0356,-965.3025
C00543=-91.901,-39.424,4.400,179.9982,0.0043,-966.7815
C00544=-92.860,-37.107,4.400,179.9983,0.0043,-968.2183
C00545=-93.786,-34.697,4.400,179.9864,0.0368,-969.6976
C00546=-94.722,-32.027,4.399,179.9239,0.2295,-971.3188
C00547=-95.617,-29.164,4.399,179.7588,0.8217,-973.0378
C00548=-96.362,-26.460,4.399,179.5542,1.7314,-974.6456
C00549=-96.890,-24.268,4.398,179.3571,2.8815,-975.9384
C00550=-97.259,-22.514,4.396,179.1610,4.2245,-976.9665
C00551=-97.591,-20.779,4.393,178.9642,5.5630,-977.9801
C00552=-97.979,-18.630,4.390,178.8252,6.7065,-979.2341
C00553=-98.490,-15.506,4.388,178.8536,7.5022,-981.0529
C00554=-99.090,-10.941,4.387,179.1355,7.8388,-983.6992
C00555=-99.524,-5.764,4.387,179.5383,7.8885,-986.6854
C00556=-99.691,0.000,4.387,-180.0000,7.8974,-990.0000
C00557=-99.524,5.764,4.387,-179.5383,7.8885,-993.3146
C00558=-99.090,10.941,4.387,-179.1355,7.8388,-996.3008
C00559=-98.490,15.506,4.388,-178.8536,7.5022,-998.9471
C00560=-97.979,18.630,4.390,-178.8252,6.7065,-1000.7659
C00561=-97.591,20.779,4.393,-178.9642,5.5630,-1002.0199
C00562=-97.259,22.514,4.396,-179.1610,4.2245,-1003.0335
C00563=-96.890,24.268,4.398,-179.3571,2.8815,-1004.0616
C00564=-96.362,26.460,4.399,-179.5542,1.7314,-1005.3544
C00565=-95.617,29.164,4.399,-179.7588,0.8217,-1006.9622
C00566=-94.722,32.027,4.399,-179.9239,0.2295,-1008.6812
C00567=-93.786,34.697,4.400,-179.9864,0.0368,-1010.3024
C00568=-92.860,37.107,4.400,-179.9983,0.0043,-1011.7817
C00569=-91.901,39.424,4.400,-179.9982,0.0043,-1013.2185
C00570=-90.851,41.782,4.400,-179.9836,0.0356,-1014.6975
C00571=-89.625,44.332,4.399,-179.8915,0.2161,-1016.3188
C00572=-88.233,46.990,4.399,-179.5895,0.7516,-1018.0383
C00573=-86.848,49.428,4.399,-179.0907,1.5395,-1019.6456
C00574=-85.672,51.352,4.398,-178.4158,2.4923,-1020.9386
C00575=-84.692,52.853,4.396,-177.6021,3.5812,-1021.9667
C00576=-83.700,54.314,4.393,-176.7898,4.6682,-1022.9801
C00577=-82.455,56.108,4.390,-176.0730,5.5771,-1024.2340
C00578=-80.608,58.679,4.388,-175.4847,6.1227,-1026.0529
C00579=-77.804,62.331,4.387,-175.0460,6.1652,-1028.6992
C00580=-74.450,66.299,4.387,-174.7278,5.9189,-1031.6856
C00581=-70.493,70.493,4.387,-174.3980,5.6020,-1035.0000
C00582=-66.299,74.450,4.387,-174.0812,5.2722,-1038.3144
C00583=-62.331,77.804,4.387,-173.8348,4.9540,-1041.3008
C00584=-58.679,80.608,4.388,-173.8773,4.5153,-1043.9471
C00585=-56.108,82.455,4.390,-174.4229,3.9270,-1045.7660
C00586=-54.314,83.700,4.393,-175.3318,3.2102,-1047.0199
C00587=-52.853,84.692,4.396,-176.4188,2.3979,-1048.0333
C00588=-51.352,85.672,4.398,-177.5077,1.5842,-1049.0614
C00589=-49.428,86.848,4.399,-178.4605,0.9093,-1050.3544
C00590=-46.990,88.233,4.399,-179.2484,0.4105,-1051.9617
C00591=-44.332,89.625,4.399,-179.7839,0.1085,-1053.6812
C00592=-41.782,90.851,4.400,-179.9644,0.0164,-1055.3025
C00593=-39.424,91.901,4.400,-179.9957,0.0018,-1056.7815
C00594=-37.107,92.860,4.400,-179.9957,0.0017,-1058.2183
C00595=-34.697,93.786,4.400,-179.9632,0.0136,-1059.6976
C00596=-32.027,94.722,4.399,-179.7705,0.0761,-1061.3188
C00597=-29.164,95.617,4.399,-179.1783,0.2412,-1063.0378
C00598=-26.460,96.362,4.399,-178.2686,0.4458,-1064.6456
C00599=-24.268,96.890,4.398,-177.1185,0.6429,-1065.9384
C00600=-22.514,97.259,4.396,-175.7755,0.8390,-1066.9665
C00601=-20.779,97.591,4.393,-174.4370,1.0358,-1067.9801
C00602=-18.630,97.979,4.390,-173.2935,1.1748,-1069.2341
C00603=-15.506,98.490,4.388,-172.4978,1.1464,-1071.0529
C00604=-10.941,99.090,4.387,-172.1612,0.8645,-1073.6992
C00605=-5.764,99.524,4.387,-172.1115,0.4617,-1076.6854
C00606=0.000,99.691,4.387,-172.1026,0.0000,-1080.0000
C00607=0.000,99.321,6.555,-168.5288,0.0000,-1080.0000
C00608=5.730,99.155,6.555,-168.5414,-0.6746,-1083.3073
C00609=10.884,98.723,6.555,-168.6119,-1.2518,-1086.2913
C00610=15.437,98.140,6.558,-169.0875,-1.6029,-1088.9391
C00611=18.547,97.668,6.566,-170.2252,-1.5293,-1090.7524
C00612=20.687,97.336,6.576,-171.8906,-1.2412,-1091.9986
C00613=22.417,97.071,6.585,-173.8606,-0.9699,-1093.0036
C00614=24.167,96.770,6.592,-175.8319,-0.7885,-1094.0220
C00615=26.351,96.303,6.595,-177.5102,-0.5868,-1095.3030
C00616=29.062,95.605,6.597,-178.8311,-0.3259,-1096.9082
C00617=31.947,94.737,6.598,-179.6815,-0.1030,-1098.6350
C00618=34.646,93.803,6.599,-179.9483,-0.0190,-1100.2716
C00619=37.090,92.867,6.600,-179.9940,-0.0024,-1101.7712
C00620=39.440,91.893,6.600,-179.9940,-0.0026,-1103.2288
C00621=41.830,90.827,6.599,-179.9500,-0.0231,-1104.7282
C00622=44.399,89.579,6.598,-179.7019,-0.1524,-1106.3649
C00623=47.053,88.152,6.597,-178.9430,-0.5962,-1108.0920
C00624=49.464,86.729,6.595,-177.8245,-1.3465,-1109.6973
C00625=51.338,85.515,6.592,-176.4942,-2.3935,-1110.9780
C00626=52.788,84.491,6.585,-174.9692,-3.6670,-1111.9962
C00627=54.199,83.455,6.576,-173.3790,-4.8831,-1113.0013
C00628=55.947,82.176,6.566,-171.9912,-5.8773,-1114.2478
C00629=58.480,80.311,6.558,-171.1269,-6.6473,-1116.0610
C00630=62.112,77.504,6.555,-171.0284,-7.2364,-1118.7088
C00631=66.061,74.165,6.555,-171.3764,-7.6887,-1121.6924
C00632=70.230,70.230,6.555,-171.8342,-8.1658,-1125.0000
C00633=74.165,66.061,6.555,-172.3113,-8.6235,-1128.3076
C00634=77.504,62.112,6.555,-172.7636,-8.9716,-1131.2912
C00635=80.311,58.480,6.558,-173.3528,-8.8731,-1133.9390
C00636=82.176,55.947,6.566,-174.1227,-8.0088,-1135.7522
C00637=83.455,54.199,6.576,-175.1169,-6.6210,-1136.9987
C00638=84.491,52.788,6.585,-176.3330,-5.0308,-1138.0038
C00639=85.515,51.338,6.592,-177.6065,-3.5058,-1139.0220
C00640=86.729,49.464,6.595,-178.6535,-2.1755,-1140.3027
C00641=88.152,47.053,6.597,-179.4038,-1.0570,-1141.9080
C00642=89.579,44.399,6.598,-179.8476,-0.2981,-1143.6351
C00643=90.827,41.830,6.599,-179.9769,-0.0500,-1145.2718
C00644=91.893,39.440,6.600,-179.9974,-0.0060,-1146.7712
C00645=92.867,37.090,6.600,-179.9976,-0.0060,-1148.2288
C00646=93.803,34.646,6.599,-179.9810,-0.0517,-1149.7284
C00647=94.737,31.947,6.598,-179.8970,-0.3185,-1151.3650
C00648=95.605,29.062,6.597,-179.6741,-1.1689,-1153.0918
C00649=96.303,26.351,6.595,-179.4132,-2.4898,-1154.6970
C00650=96.770,24.167,6.592,-179.2115,-4.1681,-1155.9780
C00651=97.071,22.417,6.585,-179.0301,-6.1394,-1156.9964
C00652=97.336,20.687,6.576,-178.7588,-8.1094,-1158.0014
C00653=97.668,18.547,6.566,-178.4707,-9.7748,-1159.2476
C00654=98.140,15.437,6.558,-178.3971,-10.9125,-1161.0609
C00655=98.723,10.884,6.555,-178.7482,-11.3881,-1163.7087
C00656=99.155,5.730,6.555,-179.3254,-11.4586,-1166.6927
C00657=99.321,0.000,6.555,180.0000,-11.4712,-1170.0000
C00658=99.155,-5.730,6.555,179.3254,-11.4585,-1173.3073
C00659=98.723,-10.884,6.555,178.7482,-11.3882,-1176.2913
C00660=98.140,-15.437,6.558,178.3971,-10.9125,-1178.9391
C00661=97.668,-18.547,6.566,178.4707,-9.7748,-1180.7524
C00662=97.336,-20.687,6.576,178.7588,-8.1094,-1181.9986
C00663=97.071,-22.417,6.585,179.0301,-6.1394,-1183.0036
C00664=96.770,-24.167,6.592,179.2115,-4.1681,-1184.0220
C00665=96.303,-26.351,6.595,179.4132,-2.4898,-1185.3030
C00666=95.605,-29.062,6.597,179.6741,-1.1689,-1186.9082
C00667=94.737,-31.947,6.598,179.8970,-0.3185,-1188.6350
C00668=93.803,-34.646,6.599,179.9810,-0.0517,-1190.2716
C00669=92.867,-37.090,6.600,179.9976,-0.0060,-1191.7712
C00670=91.893,-39.440,6.600,179.9974,-0.0060,-1193.2288
C00671=90.827,-41.830,6.599,179.9769,-0.0500,-1194.7282
C00672=89.579,-44.399,6.598,179.8476,-0.2981,-1196.3649
C00673=88.152,-47.053,6.597,179.4038,-1.0570,-1198.0920
C00674=86.729,-49.464,6.595,178.6535,-2.1755,-1199.6973
C00675=85.515,-51.338,6.592,177.6065,-3.5058,-1200.9780
C00676=84.491,-52.788,6.585,176.3330,-5.0308,-1201.9962
C00677=83.455,-54.199,6.576,175.1169,-6.6210,-1203.0013
C00678=82.176,-55.947,6.566,174.1227,-8.0088,-1204.2478
C00679=80.311,-58.480,6.558,173.3527,-8.8731,-1206.0610
C00680=77.504,-62.112,6.555,172.7636,-8.9716,-1208.7088
C00681=74.165,-66.061,6.555,172.3113,-8.6236,-1211.6924
C00682=70.230,-70.230,6.555,171.8342,-8.1658,-1215.0000
C00683=66.061,-74.165,6.555,171.3765,-7.6887,-1218.3076
C00684=62.112,-77.504,6.555,171.0284,-7.2364,-1221.2912
C00685=58.480,-80.311,6.558,171.1269,-6.6472,-1223.9390
C00686=55.947,-82.176,6.566,171.9912,-5.8773,-1225.7522
C00687=54.199,-83.455,6.576,173.3790,-4.8831,-1226.9987
C00688=52.788,-84.491,6.585,174.9692,-3.6670,-1228.0038
C00689=51.338,-85.515,6.592,176.4942,-2.3935,-1229.0220
C00690=49.464,-86.729,6.595,177.8245,-1.3465,-1230.3027
C00691=47.053,-88.152,6.597,178.9430,-0.5962,-1231.9080
C00692=44.399,-89.579,6.598,179.7019,-0.1524,-1233.6351
C00693=41.830,-90.827,6.599,179.9500,-0.0231,-1235.2718
C00694=39.440,-91.893,6.600,179.9940,-0.0026,-1236.7712
C00695=37.090,-92.867,6.600,179.9940,-0.0024,-1238.2288
C00696=34.646,-93.803,6.599,179.9483,-0.0190,-1239.7284
C00697=31.947,-94.737,6.598,179.6815,-0.1030,-1241.3650
C00698=29.062,-95.605,6.597,178.8311,-0.3259,-1243.0918
C00699=26.351,-96.303,6.595,177.5102,-0.5868,-1244.6970
C00700=24.167,-96.770,6.592,175.8319,-0.7885,-1245.9780
C00701=22.417,-97.071,6.585,173.8606,-0.9699,-1246.9964
C00702=20.687,-97.336,6.576,171.8906,-1.2412,-1248.0014
C00703=18.547,-97.668,6.566,170.2252,-1.5293,-1249.2476
C00704=15.437,-98.140,6.558,169.0875,-1.6029,-1251.0609
C00705=10.884,-98.723,6.555,168.6119,-1.2518,-1253.7087
C00706=5.730,-99.155,6.555,168.5414,-0.6746,-1256.6927
C00707=0.000,-99.321,6.555,168.5288,0.0000,-1260.0000
C00708=0.000,-99.321,6.555,168.5288,0.0000,-1260.0000
C00709=-5.730,-99.155,6.555,168.5415,0.6746,-1263.3073
C00710=-10.884,-98.723,6.555,168.6118,1.2518,-1266.2913
C00711=-15.437,-98.140,6.558,169.0875,1.6029,-1268.9391
C00712=-18.547,-97.668,6.566,170.2252,1.5293,-1270.7524
C00713=-20.687,-97.336,6.576,171.8906,1.2412,-1271.9986
C00714=-22.417,-97.071,6.585,173.8606,0.9699,-1273.0036
C00715=-24.167,-96.770,6.592,175.8319,0.7885,-1274.0220
C00716=-26.351,-96.303,6.595,177.5102,0.5868,-1275.3030
C00717=-29.062,-95.605,6.597,178.8311,0.3259,-1276.9082
C00718=-31.947,-94.737,6.598,179.6815,0.1030,-1278.6350
C00719=-34.646,-93.803,6.599,179.9483,0.0190,-1280.2716
C00720=-37.090,-92.867,6.600,179.9940,0.0024,-1281.7712
C00721=-39.440,-91.893,6.600,179.9940,0.0026,-1283.2288
C00722=-41.830,-90.827,6.599,179.9500,0.0231,-1284.7282
C00723=-44.399,-89.579,6.598,179.7019,0.1524,-1286.3649
C00724=-47.053,-88.152,6.597,178.9430,0.5962,-1288.0920
C00725=-49.464,-86.729,6.595,177.8245,1.3465,-1289.6973
C00726=-51.338,-85.515,6.592,176.4942,2.3935,-1290.9780
C00727=-52.788,-84.491,6.585,174.9692,3.6670,-1291.9962
C00728=-54.199,-83.455,6.576,173.3790,4.8831,-1293.0013
C00729=-55.947,-82.176,6.566,171.9912,5.8773,-1294.2478
C00730=-58.480,-80.311,6.558,171.1269,6.6473,-1296.0610
C00731=-62.112,-77.504,6.555,171.0284,7.2364,-1298.7088
C00732=-66.061,-74.165,6.555,171.3764,7.6887,-1301.6924
C00733=-70.230,-70.230,6.555,171.8342,8.1658,-1305.0000
C00734=-74.165,-66.061,6.555,172.3113,8.6235,-1308.3076
C00735=-77.504,-62.112,6.555,172.7636,8.9716,-1311.2912
C00736=-80.311,-58.480,6.558,173.3528,8.8731,-1313.9390
C00737=-82.176,-55.947,6.566,174.1227,8.0088,-1315.7522
C00738=-83.455,-54.199,6.576,175.1169,6.6210,-1316.9987
C00739=-84.491,-52.788,6.585,176.3330,5.0308,-1318.0038
C00740=-85.515,-51.338,6.592,177.6065,3.5058,-1319.0220
C00741=-86.729,-49.464,6.595,178.6535,2.1755,-1320.3027
C00742=-88.152,-47.053,6.597,179.4038,1.0570,-1321.9080
C00743=-89.579,-44.399,6.598,179.8476,0.2981,-1323.6351
C00744=-90.827,-41.830,6.599,179.9769,0.0500,-1325.2718
C00745=-91.893,-39.440,6.600,179.9974,0.0060,-1326.7712
C00746=-92.867,-37.090,6.600,179.9976,0.0060,-1328.2288
C00747=-93.803,-34.646,6.599,179.9810,0.0517,-1329.7284
C00748=-94.737,-31.947,6.598,179.8970,0.3185,-1331.3650
C00749=-95.605,-29.062,6.597,179.6741,1.1689,-1333.0918
C00750=-96.303,-26.351,6.595,179.4132,2.4898,-1334.6970
C00751=-96.770,-24.167,6.592,179.2115,4.1681,-1335.9780
C00752=-97.071,-22.417,6.585,179.0301,6.1394,-1336.9964
C00753=-97.336,-20.687,6.576,178.7588,8.1094,-1338.0014
C00754=-97.668,-18.547,6.566,178.4707,9.7748,-1339.2476
C00755=-98.140,-15.437,6.558,178.3971,10.9125,-1341.0609
C00756=-98.723,-10.884,6.555,178.7482,11.3881,-1343.7087
C00757=-99.155,-5.730,6.555,179.3254,11.4586,-1346.6927
C00758=-99.321,0.000,6.555,-180.0000,11.4712,-1350.0000
C00759=-99.155,5.730,6.555,-179.3254,11.4585,-1353.3073
C00760=-98.723,10.884,6.555,-178.7482,11.3882,-1356.2913
C00761=-98.140,15.437,6.558,-178.3971,10.9125,-1358.9391
C00762=-97.668,18.547,6.566,-178.4707,9.7748,-1360.7524
C00763=-97.336,20.687,6.576,-178.7588,8.1094,-1361.9986
C00764=-97.071,22.417,6.585,-179.0301,6.1394,-1363.0036
C00765=-96.770,24.167,6.592,-179.2115,4.1681,-1364.0220
C00766=-96.303,26.351,6.595,-179.4132,2.4898,-1365.3030
C00767=-95.605,29.062,6.597,-179.6741,1.1689,-1366.9082
C00768=-94.737,31.947,6.598,-179.8970,0.3185,-1368.6350
C00769=-93.803,34.646,6.599,-179.9810,0.0517,-1370.2716
C00770=-92.867,37.090,6.600,-179.9976,0.0060,-1371.7712
C00771=-91.893,39.440,6.600,-179.9974,0.0060,-1373.2288
C00772=-90.827,41.830,6.599,-179.9769,0.0500,-1374.7282
C00773=-89.579,44.399,6.598,-179.8476,0.2981,-1376.3649
C00774=-88.152,47.053,6.597,-179.4038,1.0570,-1378.0920
C00775=-86.729,49.464,6.595,-178.6535,2.1755,-1379.6973
C00776=-85.515,51.338,6.592,-177.6065,3.5058,-1380.9780
C00777=-84.491,52.788,6.585,-176.3330,5.0308,-1381.9962
C00778=-83.455,54.199,6.576,-175.1169,6.6210,-1383.0013
C00779=-82.176,55.947,6.566,-174.1227,8.0088,-1384.2478
C00780=-80.311,58.480,6.558,-173.3527,8.8731,-1386.0610
C00781=-77.504,62.112,6.555,-172.7636,8.9716,-1388.7088
C00782=-74.165,66.061,6.555,-172.3113,8.6236,-1391.6924
C00783=-70.230,70.230,6.555,-171.8342,8.1658,-1395.0000
C00784=-66.061,74.165,6.555,-171.3765,7.6887,-1398.3076
C00785=-62.112,77.504,6.555,-171.0284,7.2364,-1401.2912
C00786=-58.480,80.311,6.558,-171.1269,6.6472,-1403.9390
C00787=-55.947,82.176,6.566,-171.9912,5.8773,-1405.7522
C00788=-54.199,83.455,6.576,-173.3790,4.8831,-1406.9987
C00789=-52.788,84.491,6.585,-174.9692,3.6670,-1408.0038
C00790=-51.338,85.515,6.592,-176.4942,2.3935,-1409.0220
C00791=-49.464,86.729,6.595,-177.8245,1.3465,-1410.3027
C00792=-47.053,88.152,6.597,-178.9430,0.5962,-1411.9080
C00793=-44.399,89.579,6.598,-179.7019,0.1524,-1413.6351
C00794=-41.830,90.827,6.599,-179.9500,0.0231,-1415.2718
C00795=-39.440,91.893,6.600,-179.9940,0.0026,-1416.7712
C00796=-37.090,92.867,6.600,-179.9940,0.0024,-1418.2288
C00797=-34.646,93.803,6.599,-179.9483,0.0190,-1419.7284
C00798=-31.947,94.737,6.598,-179.6815,0.1030,-1421.3650
C00799=-29.062,95.605,6.597,-178.8311,0.3259,-1423.0918
C00800=-26.351,96.303,6.595,-177.5102,0.5868,-1424.6970
C00801=-24.167,96.770,6.592,-175.8319,0.7885,-1425.9780
C00802=-22.417,97.071,6.585,-173.8606,0.9699,-1426.9964
C00803=-20.687,97.336,6.576,-171.8906,1.2412,-1428.0014
C00804=-18.547,97.668,6.566,-170.2252,1.5293,-1429.2476
C00805=-15.437,98.140,6.558,-169.0875,1.6029,-1431.0609
C00806=-10.884,98.723,6.555,-168.6118,1.2518,-1433.7087
C00807=-5.730,99.155,6.555,-168.5415,0.6746,-1436.6927
C00808=0.000,99.321,6.555,-168.5288,0.0000,-1440.0000
C00809=0.000,98.820,8.697,-165.2395,0.0000,-1440.0000
C00810=5.684,98.656,8.697,-165.2556,-0.8746,-1443.2974
C00811=10.807,98.229,8.698,-165.3433,-1.6024,-1446.2783
C00812=15.344,97.668,8.705,-165.9346,-1.9496,-1448.9284
C00813=18.436,97.247,8.723,-167.3796,-1.6454,-1450.7347
C00814=20.563,96.991,8.745,-169.5531,-1.1205,-1451.9700
C00815=22.286,96.814,8.767,-172.1394,-0.8021,-1452.9633
C00816=24.029,96.606,8.782,-174.6912,-0.7561,-1453.9678
C00817=26.202,96.222,8.789,-176.8486,-0.6486,-1455.2327
C00818=28.922,95.588,8.792,-178.5415,-0.3776,-1456.8342
C00819=31.837,94.757,8.795,-179.6165,-0.1196,-1458.5716
C00820=34.577,93.826,8.798,-179.9364,-0.0233,-1460.2300
C00821=37.066,92.876,8.800,-179.9926,-0.0029,-1461.7565
C00822=39.463,91.883,8.800,-179.9927,-0.0031,-1463.2431
C00823=41.895,90.794,8.798,-179.9386,-0.0286,-1464.7700
C00824=44.491,89.515,8.795,-179.6442,-0.1866,-1466.4284
C00825=47.140,88.042,8.792,-178.7017,-0.7645,-1468.1658
C00826=49.511,86.567,8.789,-177.3127,-1.7714,-1469.7669
C00827=51.320,85.302,8.782,-175.7087,-3.2266,-1471.0323
C00828=52.699,84.217,8.767,-173.8629,-5.0134,-1472.0364
C00829=54.043,83.124,8.745,-171.7941,-6.6477,-1473.0299
C00830=55.728,81.800,8.723,-169.8719,-7.8577,-1474.2655
C00831=58.212,79.911,8.705,-168.6223,-8.7038,-1476.0719
C00832=61.817,77.101,8.698,-168.4305,-9.3780,-1478.7215
C00833=65.741,73.780,8.697,-168.8617,-9.9428,-1481.7023
C00834=69.877,69.877,8.697,-169.4466,-10.5535,-1485.0000
C00835=73.780,65.741,8.697,-170.0572,-11.1383,-1488.2977
C00836=77.101,61.817,8.698,-170.6220,-11.5695,-1491.2785
C00837=79.911,58.212,8.705,-171.2962,-11.3776,-1493.9281
C00838=81.800,55.728,8.723,-172.1423,-10.1281,-1495.7345
C00839=83.124,54.043,8.745,-173.3523,-8.2059,-1496.9701
C00840=84.217,52.699,8.767,-174.9866,-6.1371,-1497.9636
C00841=85.302,51.320,8.782,-176.7734,-4.2913,-1498.9677
C00842=86.567,49.511,8.789,-178.2286,-2.6873,-1500.2331
C00843=88.042,47.140,8.792,-179.2355,-1.2983,-1501.8342
C00844=89.515,44.491,8.795,-179.8134,-0.3558,-1503.5716
C00845=90.794,41.895,8.798,-179.9714,-0.0614,-1505.2300
C00846=91.883,39.463,8.800,-179.9969,-0.0073,-1506.7569
C00847=92.876,37.066,8.800,-179.9971,-0.0074,-1508.2435
C00848=93.826,34.577,8.798,-179.9767,-0.0636,-1509.7700
C00849=94.757,31.837,8.795,-179.8804,-0.3835,-1511.4284
C00850=95.588,28.922,8.792,-179.6224,-1.4585,-1513.1658
C00851=96.222,26.202,8.789,-179.3514,-3.1514,-1514.7673
C00852=96.606,24.029,8.782,-179.2439,-5.3088,-1516.0322
C00853=96.814,22.286,8.767,-179.1979,-7.8606,-1517.0367
C00854=96.991,20.563,8.745,-178.8795,-10.4469,-1518.0300
C00855=97.247,18.436,8.723,-178.3546,-12.6204,-1519.2653
C00856=97.668,15.344,8.705,-178.0504,-14.0654,-1521.0716
C00857=98.229,10.807,8.698,-178.3976,-14.6567,-1523.7217
C00858=98.656,5.684,8.697,-179.1254,-14.7444,-1526.7026
C00859=98.820,0.000,8.697,180.0000,-14.7605,-1530.0000
C00860=98.656,-5.684,8.697,179.1254,-14.7444,-1533.2974
C00861=98.229,-10.807,8.698,178.3976,-14.6567,-1536.2783
C00862=97.668,-15.344,8.705,178.0504,-14.0654,-1538.9284
C00863=97.247,-18.436,8.723,178.3546,-12.6204,-1540.7347
C00864=96.991,-20.563,8.745,178.8795,-10.4469,-1541.9700
C00865=96.814,-22.286,8.767,179.1979,-7.8606,-1542.9633
C00866=96.606,-24.029,8.782,179.2439,-5.3088,-1543.9678
C00867=96.222,-26.202,8.789,179.3514,-3.1514,-1545.2327
C00868=95.588,-28.922,8.792,179.6224,-1.4585,-1546.8342
C00869=94.757,-31.837,8.795,179.8804,-0.3835,-1548.5716
C00870=93.826,-34.577,8.798,179.9767,-0.0636,-1550.2300
C00871=92.876,-37.066,8.800,179.9971,-0.0074,-1551.7565
C00872=91.883,-39.463,8.800,179.9969,-0.0073,-1553.2431
C00873=90.794,-41.895,8.798,179.9714,-0.0614,-1554.7700
C00874=89.515,-44.491,8.795,179.8134,-0.3558,-1556.4284
C00875=88.042,-47.140,8.792,179.2355,-1.2983,-1558.1658
C00876=86.567,-49.511,8.789,178.2286,-2.6873,-1559.7669
C00877=85.302,-51.320,8.782,176.7734,-4.2913,-1561.0323
C00878=84.217,-52.699,8.767,174.9866,-6.1371,-1562.0364
C00879=83.124,-54.043,8.745,173.3523,-8.2059,-1563.0299
C00880=81.800,-55.728,8.723,172.1423,-10.1281,-1564.2655
C00881=79.911,-58.212,8.705,171.2962,-11.3777,-1566.0719
C00882=77.101,-61.817,8.698,170.6220,-11.5695,-1568.7215
C00883=73.780,-65.741,8.697,170.0572,-11.1383,-1571.7023
C00884=69.877,-69.877,8.697,169.4465,-10.5534,-1575.0000
C00885=65.741,-73.780,8.697,168.8617,-9.9428,-1578.2977
C00886=61.817,-77.101,8.698,168.4305,-9.3780,-1581.2785
C00887=58.212,-79.911,8.705,168.6224,-8.7038,-1583.9281
C00888=55.728,-81.800,8.723,169.8719,-7.8577,-1585.7345
C00889=54.043,-83.124,8.745,171.7941,-6.6477,-1586.9701
C00890=52.699,-84.217,8.767,173.8629,-5.0134,-1587.9636
C00891=51.320,-85.302,8.782,175.7087,-3.2266,-1588.9677
C00892=49.511,-86.567,8.789,177.3127,-1.7714,-1590.2331
C00893=47.140,-88.042,8.792,178.7017,-0.7645,-1591.8342
C00894=44.491,-89.515,8.795,179.6442,-0.1866,-1593.5716
C00895=41.895,-90.794,8.798,179.9386,-0.0286,-1595.2300
C00896=39.463,-91.883,8.800,179.9927,-0.0031,-1596.7569
C00897=37.066,-92.876,8.800,179.9926,-0.0029,-1598.2435
C00898=34.577,-93.826,8.798,179.9364,-0.0233,-1599.7700
C00899=31.837,-94.757,8.795,179.6165,-0.1196,-1601.4284
C00900=28.922,-95.588,8.792,178.5415,-0.3776,-1603.1658
C00901=26.202,-96.222,8.789,176.8486,-0.6486,-1604.7673
C00902=24.029,-96.606,8.782,174.6912,-0.7561,-1606.0322
C00903=22.286,-96.814,8.767,172.1394,-0.8021,-1607.0367
C00904=20.563,-96.991,8.745,169.5531,-1.1205,-1608.0300
C00905=18.436,-97.247,8.723,167.3796,-1.6454,-1609.2653
C00906=15.344,-97.668,8.705,165.9346,-1.9496,-1611.0716
C00907=10.807,-98.229,8.698,165.3433,-1.6024,-1613.7217
C00908=5.684,-98.656,8.697,165.2556,-0.8746,-1616.7026
C00909=0.000,-98.820,8.697,165.2395,0.0000,-1620.0000
C00910=0.000,-98.820,8.697,165.2395,0.0000,-1620.0000
C00911=-5.684,-98.656,8.697,165.2556,0.8746,-1623.2974
C00912=-10.807,-98.229,8.698,165.3433,1.6024,-1626.2783
C00913=-15.344,-97.668,8.705,165.9346,1.9496,-1628.9284
C00914=-18.436,-97.247,8.723,167.3796,1.6454,-1630.7347
C00915=-20.563,-96.991,8.745,169.5531,1.1205,-1631.9700
C00916=-22.286,-96.814,8.767,172.1394,0.8021,-1632.9633
C00917=-24.029,-96.606,8.782,174.6912,0.7561,-1633.9678
C00918=-26.202,-96.222,8.789,176.8486,0.6486,-1635.2327
C00919=-28.922,-95.588,8.792,178.5415,0.3776,-1636.8342
C00920=-31.837,-94.757,8.795,179.6165,0.1196,-1638.5716
C00921=-34.577,-93.826,8.798,179.9364,0.0233,-1640.2300
C00922=-37.066,-92.876,8.800,179.9926,0.0029,-1641.7565
C00923=-39.463,-91.883,8.800,179.9927,0.0031,-1643.2431
C00924=-41.895,-90.794,8.798,179.9386,0.0286,-1644.7700
C00925=-44.491,-89.515,8.795,179.6442,0.1866,-1646.4284
C00926=-47.140,-88.042,8.792,178.7017,0.7645,-1648.1658
C00927=-49.511,-86.567,8.789,177.3127,1.7714,-1649.7669
C00928=-51.320,-85.302,8.782,175.7087,3.2266,-1651.0323
C00929=-52.699,-84.217,8.767,173.8629,5.0134,-1652.0364
C00930=-54.043,-83.124,8.745,171.7941,6.6477,-1653.0299
C00931=-55.728,-81.800,8.723,169.8719,7.8577,-1654.2655
C00932=-58.212,-79.911,8.705,168.6223,8.7038,-1656.0719
C00933=-61.817,-77.101,8.698,168.4305,9.3780,-1658.7215
C00934=-65.741,-73.780,8.697,168.8617,9.9428,-1661.7023
C00935=-69.877,-69.877,8.697,169.4466,10.5535,-1665.0000
C00936=-73.780,-65.741,8.697,170.0572,11.1383,-1668.2977
C00937=-77.101,-61.817,8.698,170.6220,11.5695,-1671.2785
C00938=-79.911,-58.212,8.705,171.2962,11.3776,-1673.9281
C00939=-81.800,-55.728,8.723,172.1423,10.1281,-1675.7345
C00940=-83.124,-54.043,8.745,173.3523,8.2059,-1676.9701
C00941=-84.217,-52.699,8.767,174.9866,6.1371,-1677.9636
C00942=-85.302,-51.320,8.782,176.7734,4.2913,-1678.9677
C00943=-86.567,-49.511,8.789,178.2286,2.6873,-1680.2331
C00944=-88.042,-47.140,8.792,179.2355,1.2983,-1681.8342
C00945=-89.515,-44.491,8.795,179.8134,0.3558,-1683.5716
C00946=-90.794,-41.895,8.798,179.9714,0.0614,-1685.2300
C00947=-91.883,-39.463,8.800,179.9969,0.0073,-1686.7569
C00948=-92.876,-37.066,8.800,179.9971,0.0074,-1688.2435
C00949=-93.826,-34.577,8.798,179.9767,0.0636,-1689.7700
C00950=-94.757,-31.837,8.795,179.8804,0.3835,-1691.4284
C00951=-95.588,-28.922,8.792,179.6224,1.4585,-1693.1658
C00952=-96.222,-26.202,8.789,179.3514,3.1514,-1694.7673
C00953=-96.606,-24.029,8.782,179.2439,5.3088,-1696.0322
C00954=-96.814,-22.286,8.767,179.1979,7.8606,-1697.0367
C00955=-96.991,-20.563,8.745,178.8795,10.4469,-1698.0300
C00956=-97.247,-18.436,8.723,178.3546,12.6204,-1699.2653
C00957=-97.668,-15.344,8.705,178.0504,14.0654,-1701.0716
C00958=-98.229,-10.807,8.698,178.3976,14.6567,-1703.7217
C00959=-98.656,-5.684,8.697,179.1254,14.7444,-1706.7026
C00960=-98.820,0.000,8.697,-180.0000,14.7605,-1710.0000
C00961=-98.656,5.684,8.697,-179.1254,14.7444,-1713.2974
C00962=-98.229,10.807,8.698,-178.3976,14.6567,-1716.2783
C00963=-97.668,15.344,8.705,-178.0504,14.0654,-1718.9284
C00964=-97.247,18.436,8.723,-178.3546,12.6204,-1720.7347
C00965=-96.991,20.563,8.745,-178.8795,10.4469,-1721.9700
C00966=-96.814,22.286,8.767,-179.1979,7.8606,-1722.9633
C00967=-96.606,24.029,8.782,-179.2439,5.3088,-1723.9678
C00968=-96.222,26.202,8.789,-179.3514,3.1514,-1725.2327
C00969=-95.588,28.922,8.792,-179.6224,1.4585,-1726.8342
C00970=-94.757,31.837,8.795,-179.8804,0.3835,-1728.5716
C00971=-93.826,34.577,8.798,-179.9767,0.0636,-1730.2300
C00972=-92.876,37.066,8.800,-179.9971,0.0074,-1731.7565
C00973=-91.883,39.463,8.800,-179.9969,0.0073,-1733.2431
C00974=-90.794,41.895,8.798,-179.9714,0.0614,-1734.7700
C00975=-89.515,44.491,8.795,-179.8134,0.3558,-1736.4284
C00976=-88.042,47.140,8.792,-179.2355,1.2983,-1738.1658
C00977=-86.567,49.511,8.789,-178.2286,2.6873,-1739.7669
C00978=-85.302,51.320,8.782,-176.7734,4.2913,-1741.0323
C00979=-84.217,52.699,8.767,-174.9866,6.1371,-1742.0364
C00980=-83.124,54.043,8.745,-173.3523,8.2059,-1743.0299
C00981=-81.800,55.728,8.723,-172.1423,10.1281,-1744.2655
C00982=-79.911,58.212,8.705,-171.2962,11.3777,-1746.0719
C00983=-77.101,61.817,8.698,-170.6220,11.5695,-1748.7215
C00984=-73.780,65.741,8.697,-170.0572,11.1383,-1751.7023
C00985=-69.877,69.877,8.697,-169.4465,10.5534,-1755.0000
C00986=-65.741,73.780,8.697,-168.8617,9.9428,-1758.2977
C00987=-61.817,77.101,8.698,-168.4305,9.3780,-1761.2785
C00988=-58.212,79.911,8.705,-168.6224,8.7038,-1763.9281
C00989=-55.728,81.800,8.723,-169.8719,7.8577,-1765.7345
C00990=-54.043,83.124,8.745,-171.7941,6.6477,-1766.9701
C00991=-52.699,84.217,8.767,-173.8629,5.0134,-1767.9636
C00992=-51.320,85.302,8.782,-175.7087,3.2266,-1768.9677
C00993=-49.511,86.567,8.789,-177.3127,1.7714,-1770.2331
C00994=-47.140,88.042,8.792,-178.7017,0.7645,-1771.8342
C00995=-44.491,89.515,8.795,-179.6442,0.1866,-1773.5716
C00996=-41.895,90.794,8.798,-179.9386,0.0286,-1775.2300
C00997=-39.463,91.883,8.800,-179.9927,0.0031,-1776.7569
C00998=-37.066,92.876,8.800,-179.9926,0.0029,-1778.2435
C00999=-34.577,93.826,8.798,-179.9364,0.0233,-1779.7700
C01000=-31.837,94.757,8.795,-179.6165,0.1196,-1781.4284
C01001=-28.922,95.588,8.792,-178.5415,0.3776,-1783.1658
C01002=-26.202,96.222,8.789,-176.8486,0.6486,-1784.7673
C01003=-24.029,96.606,8.782,-174.6912,0.7561,-1786.0322
C01004=-22.286,96.814,8.767,-172.1394,0.8021,-1787.0367
C01005=-20.563,96.991,8.745,-169.5531,1.1205,-1788.0300
C01006=-18.436,97.247,8.723,-167.3796,1.6454,-1789.2653
C01007=-15.344,97.668,8.705,-165.9346,1.9496,-1791.0716
C01008=-10.807,98.229,8.698,-165.3433,1.6024,-1793.7217
C01009=-5.684,98.656,8.697,-165.2556,0.8746,-1796.7026
C01010=0.000,98.820,8.697,-165.2395,0.0000,-1800.0000
C01011=0.000,98.204,10.809,-162.2405,0.0001,-1800.0000
C01012=5.628,98.041,10.809,-162.2594,-1.0613,-1803.2854
C01013=10.712,97.620,10.809,-162.3610,-1.9132,-1806.2621
C01014=15.229,97.084,10.823,-163.0467,-2.1695,-1808.9150
C01015=18.298,96.727,10.856,-164.7843,-1.4750,-1810.7121
C01016=20.409,96.562,10.898,-167.4920,-0.6133,-1811.9342
C01017=22.123,96.495,10.937,-170.6949,-0.2914,-1812.9128
C01018=23.856,96.400,10.965,-173.7465,-0.5203,-1813.8997
C01019=26.016,96.121,10.978,-176.3051,-0.6217,-1815.1448
C01020=28.748,95.567,10.985,-178.3192,-0.3939,-1816.7421
C01021=31.699,94.782,10.991,-179.5791,-0.1255,-1818.4921
C01022=34.490,93.854,10.996,-179.9278,-0.0262,-1820.1777
C01023=37.037,92.887,11.000,-179.9917,-0.0033,-1821.7387
C01024=39.492,91.870,11.000,-179.9918,-0.0035,-1823.2613
C01025=41.977,90.753,10.996,-179.9305,-0.0325,-1824.8225
C01026=44.606,89.436,10.991,-179.6137,-0.2089,-1826.5076
C01027=47.248,87.904,10.985,-178.5329,-0.9103,-1828.2578
C01028=49.571,86.364,10.978,-176.9470,-2.1756,-1829.8549
C01029=51.296,85.034,10.965,-175.2038,-4.0647,-1831.1001
C01030=52.589,83.875,10.937,-173.1881,-6.4053,-1832.0874
C01031=53.849,82.711,10.898,-170.6621,-8.4913,-1833.0661
C01032=55.458,81.334,10.856,-168.1110,-9.8772,-1834.2883
C01033=57.880,79.417,10.823,-166.3774,-10.6897,-1836.0850
C01034=61.453,76.603,10.809,-166.0469,-11.3770,-1838.7375
C01035=65.346,73.305,10.809,-166.5413,-12.0309,-1841.7146
C01036=69.440,69.440,10.809,-167.2392,-12.7609,-1845.0000
C01037=73.305,65.346,10.809,-167.9691,-13.4586,-1848.2854
C01038=76.603,61.453,10.809,-168.6230,-13.9530,-1851.2625
C01039=79.417,57.880,10.823,-169.3103,-13.6226,-1853.9150
C01040=81.334,55.458,10.856,-170.1228,-11.8890,-1855.7117
C01041=82.711,53.849,10.898,-171.5087,-9.3379,-1856.9339
C01042=83.875,52.589,10.937,-173.5947,-6.8119,-1857.9126
C01043=85.034,51.296,10.965,-175.9353,-4.7962,-1858.8999
C01044=86.364,49.571,10.978,-177.8244,-3.0530,-1860.1451
C01045=87.904,47.248,10.985,-179.0897,-1.4671,-1861.7422
C01046=89.436,44.606,10.991,-179.7911,-0.3863,-1863.4924
C01047=90.753,41.977,10.996,-179.9675,-0.0695,-1865.1775
C01048=91.870,39.492,11.000,-179.9965,-0.0082,-1866.7387
C01049=92.887,37.037,11.000,-179.9967,-0.0083,-1868.2613
C01050=93.854,34.490,10.996,-179.9738,-0.0722,-1869.8223
C01051=94.782,31.699,10.991,-179.8745,-0.4209,-1871.5079
C01052=95.567,28.748,10.985,-179.6061,-1.6808,-1873.2579
C01053=96.121,26.016,10.978,-179.3783,-3.6949,-1874.8552
C01054=96.400,23.856,10.965,-179.4797,-6.2535,-1876.1003
C01055=96.495,22.123,10.937,-179.7086,-9.3051,-1877.0872
C01056=96.562,20.409,10.898,-179.3867,-12.5080,-1878.0658
C01057=96.727,18.298,10.856,-178.5250,-15.2157,-1879.2879
C01058=97.084,15.229,10.823,-177.8305,-16.9533,-1881.0850
C01059=97.620,10.712,10.809,-178.0868,-17.6390,-1883.7379
C01060=98.041,5.628,10.809,-178.9387,-17.7406,-1886.7146
C01061=98.204,0.000,10.809,179.9999,-17.7595,-1890.0000
C01062=98.041,-5.628,10.809,178.9388,-17.7405,-1893.2854
C01063=97.620,-10.712,10.809,178.0869,-17.6390,-1896.2621
C01064=97.084,-15.229,10.823,177.8304,-16.9533,-1898.9150
C01065=96.727,-18.298,10.856,178.5250,-15.2157,-1900.7121
C01066=96.562,-20.409,10.898,179.3867,-12.5080,-1901.9342
C01067=96.495,-22.123,10.937,179.7086,-9.3051,-1902.9128
C01068=96.400,-23.856,10.965,179.4797,-6.2535,-1903.8997
C01069=96.121,-26.016,10.978,179.3783,-3.6949,-1905.1448
C01070=95.567,-28.748,10.985,179.6061,-1.6808,-1906.7421
C01071=94.782,-31.699,10.991,179.8745,-0.4209,-1908.4921
C01072=93.854,-34.490,10.996,179.9738,-0.0722,-1910.1777
C01073=92.887,-37.037,11.000,179.9967,-0.0083,-1911.7387
C01074=91.870,-39.492,11.000,179.9965,-0.0082,-1913.2613
C01075=90.753,-41.977,10.996,179.9675,-0.0695,-1914.8225
C01076=89.436,-44.606,10.991,179.7911,-0.3863,-1916.5076
C01077=87.904,-47.248,10.985,179.0897,-1.4671,-1918.2578
C01078=86.364,-49.571,10.978,177.8244,-3.0530,-1919.8549
C01079=85.034,-51.296,10.965,175.9353,-4.7962,-1921.1001
C01080=83.875,-52.589,10.937,173.5947,-6.8119,-1922.0874
C01081=82.711,-53.849,10.898,171.5087,-9.3379,-1923.0661
C01082=81.334,-55.458,10.856,170.1228,-11.8890,-1924.2883
C01083=79.417,-57.880,10.823,169.3103,-13.6226,-1926.0850
C01084=76.603,-61.453,10.809,168.6230,-13.9531,-1928.7375
C01085=73.305,-65.346,10.809,167.9691,-13.4587,-1931.7146
C01086=69.440,-69.440,10.809,167.2391,-12.7608,-1935.0000
C01087=65.346,-73.305,10.809,166.5414,-12.0309,-1938.2854
C01088=61.453,-76.603,10.809,166.0470,-11.3770,-1941.2625
C01089=57.880,-79.417,10.823,166.3774,-10.6897,-1943.9150
C01090=55.458,-81.334,10.856,168.1110,-9.8772,-1945.7117
C01091=53.849,-82.711,10.898,170.6621,-8.4913,-1946.9339
C01092=52.589,-83.875,10.937,173.1881,-6.4053,-1947.9126
C01093=51.296,-85.034,10.965,175.2038,-4.0647,-1948.8999
C01094=49.571,-86.364,10.978,176.9470,-2.1756,-1950.1451
C01095=47.248,-87.904,10.985,178.5329,-0.9103,-1951.7422
C01096=44.606,-89.436,10.991,179.6137,-0.2089,-1953.4924
C01097=41.977,-90.753,10.996,179.9305,-0.0325,-1955.1775
C01098=39.492,-91.870,11.000,179.9918,-0.0035,-1956.7387
C01099=37.037,-92.887,11.000,179.9917,-0.0033,-1958.2613
C01100=34.490,-93.854,10.996,179.9278,-0.0262,-1959.8223
C01101=31.699,-94.782,10.991,179.5791,-0.1255,-1961.5079
C01102=28.748,-95.567,10.985,178.3192,-0.3939,-1963.2579
C01103=26.016,-96.121,10.978,176.3051,-0.6217,-1964.8552
C01104=23.856,-96.400,10.965,173.7465,-0.5203,-1966.1003
C01105=22.123,-96.495,10.937,170.6949,-0.2914,-1967.0872
C01106=20.409,-96.562,10.898,167.4920,-0.6133,-1968.0658
C01107=18.298,-96.727,10.856,164.7843,-1.4750,-1969.2879
C01108=15.229,-97.084,10.823,163.0467,-2.1695,-1971.0850
C01109=10.712,-97.620,10.809,162.3610,-1.9132,-1973.7379
C01110=5.628,-98.041,10.809,162.2594,-1.0613,-1976.7146
C01111=0.000,-98.204,10.809,162.2405,0.0001,-1980.0000
C01112=0.000,-98.204,10.809,162.2405,0.0001,-1980.0000
C01113=-5.628,-98.041,10.809,162.2595,1.0612,-1983.2854
C01114=-10.712,-97.620,10.809,162.3610,1.9131,-1986.2621
C01115=-15.229,-97.084,10.823,163.0467,2.1696,-1988.9150
C01116=-18.298,-96.727,10.856,164.7843,1.4750,-1990.7121
C01117=-20.409,-96.562,10.898,167.4920,0.6133,-1991.9342
C01118=-22.123,-96.495,10.937,170.6949,0.2914,-1992.9128
C01119=-23.856,-96.400,10.965,173.7465,0.5203,-1993.8997
C01120=-26.016,-96.121,10.978,176.3051,0.6217,-1995.1448
C01121=-28.748,-95.567,10.985,178.3192,0.3939,-1996.7421
C01122=-31.699,-94.782,10.991,179.5791,0.1255,-1998.4921
C01123=-34.490,-93.854,10.996,179.9278,0.0262,-2000.1777
C01124=-37.037,-92.887,11.000,179.9917,0.0033,-2001.7387
C01125=-39.492,-91.870,11.000,179.9918,0.0035,-2003.2613
C01126=-41.977,-90.753,10.996,179.9305,0.0325,-2004.8225
C01127=-44.606,-89.436,10.991,179.6137,0.2089,-2006.5076
C01128=-47.248,-87.904,10.985,178.5329,0.9103,-2008.2578
C01129=-49.571,-86.364,10.978,176.9470,2.1756,-2009.8549
C01130=-51.296,-85.034,10.965,175.2038,4.0647,-2011.1001
C01131=-52.589,-83.875,10.937,173.1881,6.4053,-2012.0874
C01132=-53.849,-82.711,10.898,170.6621,8.4913,-2013.0661
C01133=-55.458,-81.334,10.856,168.1110,9.8772,-2014.2883
C01134=-57.880,-79.417,10.823,166.3774,10.6897,-2016.0850
C01135=-61.453,-76.603,10.809,166.0469,11.3770,-2018.7375
C01136=-65.346,-73.305,10.809,166.5413,12.0309,-2021.7146
C01137=-69.440,-69.440,10.809,167.2392,12.7609,-2025.0000
C01138=-73.305,-65.346,10.809,167.9691,13.4586,-2028.2854
C01139=-76.603,-61.453,10.809,168.6230,13.9530,-2031.2625
C01140=-79.417,-57.880,10.823,169.3103,13.6226,-2033.9150
C01141=-81.334,-55.458,10.856,170.1228,11.8890,-2035.7117
C01142=-82.711,-53.849,10.898,171.5087,9.3379,-2036.9339
C01143=-83.875,-52.589,10.937,173.5947,6.8119,-2037.9126
C01144=-85.034,-51.296,10.965,175.9353,4.7962,-2038.8999
C01145=-86.364,-49.571,10.978,177.8244,3.0530,-2040.1451
C01146=-87.904,-47.248,10.985,179.0897,1.4671,-2041.7422
C01147=-89.436,-44.606,10.991,179.7911,0.3863,-2043.4924
C01148=-90.753,-41.977,10.996,179.9675,0.0695,-2045.1775
C01149=-91.870,-39.492,11.000,179.9965,0.0082,-2046.7387
C01150=-92.887,-37.037,11.000,179.9967,0.0083,-2048.2613
C01151=-93.854,-34.490,10.996,179.9738,0.0722,-2049.8223
C01152=-94.782,-31.699,10.991,179.8745,0.4209,-2051.5079
C01153=-95.567,-28.748,10.985,179.6061,1.6808,-2053.2579
C01154=-96.121,-26.016,10.978,179.3783,3.6949,-2054.8552
C01155=-96.400,-23.856,10.965,179.4797,6.2535,-2056.1003
C01156=-96.495,-22.123,10.937,179.7086,9.3051,-2057.0872
C01157=-96.562,-20.409,10.898,179.3867,12.5080,-2058.0658
C01158=-96.727,-18.298,10.856,178.5250,15.2157,-2059.2879
C01159=-97.084,-15.229,10.823,177.8305,16.9533,-2061.0850
C01160=-97.620,-10.712,10.809,178.0868,17.6390,-2063.7379
C01161=-98.041,-5.628,10.809,178.9387,17.7406,-2066.7146
C01162=-98.204,0.000,10.809,-179.9999,17.7595,-2070.0000
C01163=-98.041,5.628,10.809,-178.9388,17.7405,-2073.2854
C01164=-97.620,10.712,10.809,-178.0869,17.6390,-2076.2621
C01165=-97.084,15.229,10.823,-177.8304,16.9533,-2078.9150
C01166=-96.727,18.298,10.856,-178.5250,15.2157,-2080.7121
C01167=-96.562,20.409,10.898,-179.3867,12.5080,-2081.9342
C01168=-96.495,22.123,10.937,-179.7086,9.3051,-2082.9128
C01169=-96.400,23.856,10.965,-179.4797,6.2535,-2083.8997
C01170=-96.121,26.016,10.978,-179.3783,3.6949,-2085.1448
C01171=-95.567,28.748,10.985,-179.6061,1.6808,-2086.7421
C01172=-94.782,31.699,10.991,-179.8745,0.4209,-2088.4921
C01173=-93.854,34.490,10.996,-179.9738,0.0722,-2090.1777
C01174=-92.887,37.037,11.000,-179.9967,0.0083,-2091.7387
C01175=-91.870,39.492,11.000,-179.9965,0.0082,-2093.2613
C01176=-90.753,41.977,10.996,-179.9675,0.0695,-2094.8225
C01177=-89.436,44.606,10.991,-179.7911,0.3863,-2096.5076
C01178=-87.904,47.248,10.985,-179.0897,1.4671,-2098.2578
C01179=-86.364,49.571,10.978,-177.8244,3.0530,-2099.8549
C01180=-85.034,51.296,10.965,-175.9353,4.7962,-2101.1001
C01181=-83.875,52.589,10.937,-173.5947,6.8119,-2102.0874
C01182=-82.711,53.849,10.898,-171.5087,9.3379,-2103.0661
C01183=-81.334,55.458,10.856,-170.1228,11.8890,-2104.2883
C01184=-79.417,57.880,10.823,-169.3103,13.6226,-2106.0850
C01185=-76.603,61.453,10.809,-168.6230,13.9531,-2108.7375
C01186=-73.305,65.346,10.809,-167.9691,13.4587,-2111.7146
C01187=-69.440,69.440,10.809,-167.2391,12.7608,-2115.0000
C01188=-65.346,73.305,10.809,-166.5414,12.0309,-2118.2854
C01189=-61.453,76.603,10.809,-166.0470,11.3770,-2121.2625
C01190=-57.880,79.417,10.823,-166.3774,10.6897,-2123.9150
C01191=-55.458,81.334,10.856,-168.1110,9.8772,-2125.7117
C01192=-53.849,82.711,10.898,-170.6621,8.4913,-2126.9339
C01193=-52.589,83.875,10.937,-173.1881,6.4053,-2127.9126
C01194=-51.296,85.034,10.965,-175.2038,4.0647,-2128.8999
C01195=-49.571,86.364,10.978,-176.9470,2.1756,-2130.1451
C01196=-47.248,87.904,10.985,-178.5329,0.9103,-2131.7422
C01197=-44.606,89.436,10.991,-179.6137,0.2089,-2133.4924
C01198=-41.977,90.753,10.996,-179.9305,0.0325,-2135.1775
C01199=-39.492,91.870,11.000,-179.9918,0.0035,-2136.7387
C01200=-37.037,92.887,11.000,-179.9917,0.0033,-2138.2613
C01201=-34.490,93.854,10.996,-179.9278,0.0262,-2139.8223
C01202=-31.699,94.782,10.991,-179.5791,0.1255,-2141.5079
C01203=-28.748,95.567,10.985,-178.3192,0.3939,-2143.2579
C01204=-26.016,96.121,10.978,-176.3051,0.6217,-2144.8552
C01205=-23.856,96.400,10.965,-173.7465,0.5203,-2146.1003
C01206=-22.123,96.495,10.937,-170.6949,0.2914,-2147.0872
C01207=-20.409,96.562,10.898,-167.4920,0.6133,-2148.0658
C01208=-18.298,96.727,10.856,-164.7843,1.4750,-2149.2879
C01209=-15.229,97.084,10.823,-163.0467,2.1696,-2151.0850
C01210=-10.712,97.620,10.809,-162.3610,1.9131,-2153.7379
C01211=-5.628,98.041,10.809,-162.2595,1.0612,-2156.7146
C01212=0.000,98.204,10.809,-162.2405,0.0001,-2160.0000
C01213=0.000,97.482,12.888,-159.5253,0.0001,-2160.0000
C01214=5.562,97.322,12.887,-159.5467,-1.2345,-2163.2709
C01215=10.602,96.908,12.888,-159.6590,-2.1823,-2166.2435
C01216=15.094,96.401,12.910,-160.4230,-2.2510,-2168.8988
C01217=18.135,96.115,12.963,-162.4714,-0.9834,-2170.6850
C01218=20.227,96.057,13.031,-165.7975,0.3024,-2171.8912
C01219=21.929,96.117,13.096,-169.6348,0.5559,-2172.8520
C01220=23.652,96.157,13.142,-173.0616,-0.0823,-2173.8189
C01221=25.795,96.000,13.164,-175.9036,-0.5053,-2175.0400
C01222=28.540,95.542,13.175,-178.1724,-0.3760,-2176.6318
C01223=31.535,94.812,13.184,-179.5717,-0.1209,-2178.3974
C01224=34.387,93.888,13.193,-179.9229,-0.0278,-2180.1155
C01225=37.002,92.901,13.199,-179.9912,-0.0035,-2181.7171
C01226=39.526,91.855,13.199,-179.9913,-0.0038,-2183.2826
C01227=42.074,90.704,13.193,-179.9258,-0.0349,-2184.8847
C01228=44.743,89.341,13.184,-179.6117,-0.2174,-2186.6022
C01229=47.377,87.740,13.175,-178.4418,-1.0268,-2188.3677
C01230=49.643,86.123,13.164,-176.7447,-2.5426,-2189.9600
C01231=51.269,84.717,13.142,-175.0240,-4.8604,-2191.1815
C01232=52.459,83.471,13.096,-173.0176,-7.7557,-2192.1481
C01233=53.620,82.225,13.031,-170.0612,-10.3532,-2193.1089
C01234=55.140,80.787,12.963,-166.7496,-11.9257,-2194.3149
C01235=57.492,78.839,12.910,-164.3969,-12.6081,-2196.1008
C01236=61.028,76.021,12.888,-163.8761,-13.2352,-2198.7567
C01237=64.884,72.750,12.887,-164.4132,-13.9544,-2201.7290
C01238=68.930,68.930,12.888,-165.2103,-14.7899,-2205.0000
C01239=72.750,64.884,12.887,-166.0456,-15.5867,-2208.2710
C01240=76.021,61.028,12.888,-166.7646,-16.1238,-2211.2433
C01241=78.839,57.492,12.910,-167.3920,-15.6031,-2213.8992
C01242=80.787,55.140,12.963,-168.0743,-13.2504,-2215.6851
C01243=82.225,53.620,13.031,-169.6468,-9.9388,-2216.8911
C01244=83.471,52.459,13.096,-172.2443,-6.9824,-2217.8519
C01245=84.717,51.269,13.142,-175.1396,-4.9760,-2218.8185
C01246=86.123,49.643,13.164,-177.4574,-3.2553,-2220.0400
C01247=87.740,47.377,13.175,-178.9732,-1.5582,-2221.6323
C01248=89.341,44.743,13.184,-179.7826,-0.3883,-2223.3978
C01249=90.704,42.074,13.193,-179.9651,-0.0742,-2225.1153
C01250=91.855,39.526,13.199,-179.9962,-0.0087,-2226.7174
C01251=92.901,37.002,13.199,-179.9965,-0.0088,-2228.2829
C01252=93.888,34.387,13.193,-179.9722,-0.0771,-2229.8845
C01253=94.812,31.535,13.184,-179.8791,-0.4283,-2231.6026
C01254=95.542,28.540,13.175,-179.6240,-1.8276,-2233.3682
C01255=96.000,25.795,13.164,-179.4947,-4.0964,-2234.9600
C01256=96.157,23.652,13.142,-179.9177,-6.9384,-2236.1811
C01257=96.117,21.929,13.096,179.4441,-10.3652,-2237.1480
C01258=96.057,20.227,13.031,179.6976,-14.2025,-2238.1088
C01259=96.115,18.135,12.963,-179.0166,-17.5286,-2239.3150
C01260=96.401,15.094,12.910,-177.7490,-19.5770,-2241.1012
C01261=96.908,10.602,12.888,-177.8177,-20.3410,-2243.7565
C01262=97.322,5.562,12.887,-178.7655,-20.4533,-2246.7291
C01263=97.482,0.000,12.888,179.9999,-20.4747,-2250.0000
C01264=97.322,-5.562,12.887,178.7657,-20.4533,-2253.2709
C01265=96.908,-10.602,12.888,177.8179,-20.3410,-2256.2435
C01266=96.401,-15.094,12.910,177.7489,-19.5769,-2258.8988
C01267=96.115,-18.135,12.963,179.0166,-17.5286,-2260.6850
C01268=96.057,-20.227,13.031,-179.6976,-14.2025,-2261.8912
C01269=96.117,-21.929,13.096,-179.4441,-10.3652,-2262.8520
C01270=96.157,-23.652,13.142,179.9177,-6.9384,-2263.8189
C01271=96.000,-25.795,13.164,179.4947,-4.0964,-2265.0400
C01272=95.542,-28.540,13.175,179.6240,-1.8276,-2266.6318
C01273=94.812,-31.535,13.184,179.8791,-0.4283,-2268.3974
C01274=93.888,-34.387,13.193,179.9722,-0.0771,-2270.1155
C01275=92.901,-37.002,13.199,179.9965,-0.0088,-2271.7171
C01276=91.855,-39.526,13.199,179.9962,-0.0087,-2273.2826
C01277=90.704,-42.074,13.193,179.9651,-0.0742,-2274.8847
C01278=89.341,-44.743,13.184,179.7826,-0.3883,-2276.6022
C01279=87.740,-47.377,13.175,178.9732,-1.5582,-2278.3677
C01280=86.123,-49.643,13.164,177.4574,-3.2553,-2279.9600
C01281=84.717,-51.269,13.142,175.1396,-4.9760,-2281.1815
C01282=83.471,-52.459,13.096,172.2443,-6.9824,-2282.1481
C01283=82.225,-53.620,13.031,169.6468,-9.9388,-2283.1089
C01284=80.787,-55.140,12.963,168.0743,-13.2504,-2284.3149
C01285=78.839,-57.492,12.910,167.3919,-15.6031,-2286.1008
C01286=76.021,-61.028,12.888,166.7648,-16.1239,-2288.7567
C01287=72.750,-64.884,12.887,166.0456,-15.5868,-2291.7290
C01288=68.930,-68.930,12.888,165.2101,-14.7897,-2295.0000
C01289=64.884,-72.750,12.887,164.4133,-13.9544,-2298.2710
C01290=61.028,-76.021,12.888,163.8762,-13.2354,-2301.2433
C01291=57.492,-78.839,12.910,164.3969,-12.6080,-2303.8992
C01292=55.140,-80.787,12.963,166.7496,-11.9257,-2305.6851
C01293=53.620,-82.225,13.031,170.0612,-10.3532,-2306.8911
C01294=52.459,-83.471,13.096,173.0176,-7.7557,-2307.8519
C01295=51.269,-84.717,13.142,175.0240,-4.8604,-2308.8185
C01296=49.643,-86.123,13.164,176.7447,-2.5426,-2310.0400
C01297=47.377,-87.740,13.175,178.4418,-1.0268,-2311.6323
C01298=44.743,-89.341,13.184,179.6117,-0.2174,-2313.3978
C01299=42.074,-90.704,13.193,179.9258,-0.0349,-2315.1153
C01300=39.526,-91.855,13.199,179.9913,-0.0038,-2316.7174
C01301=37.002,-92.901,13.199,179.9912,-0.0035,-2318.2829
C01302=34.387,-93.888,13.193,179.9229,-0.0278,-2319.8845
C01303=31.535,-94.812,13.184,179.5717,-0.1209,-2321.6026
C01304=28.540,-95.542,13.175,178.1724,-0.3760,-2323.3682
C01305=25.795,-96.000,13.164,175.9036,-0.5053,-2324.9600
C01306=23.652,-96.157,13.142,173.0616,-0.0823,-2326.1811
C01307=21.929,-96.117,13.096,169.6348,0.5559,-2327.1480
C01308=20.227,-96.057,13.031,165.7975,0.3024,-2328.1088
C01309=18.135,-96.115,12.963,162.4714,-0.9834,-2329.3150
C01310=15.094,-96.401,12.910,160.4230,-2.2510,-2331.1012
C01311=10.602,-96.908,12.888,159.6590,-2.1823,-2333.7565
C01312=5.562,-97.322,12.887,159.5467,-1.2345,-2336.7291
C01313=0.000,-97.482,12.888,159.5253,0.0001,-2340.0000
C01314=0.000,-97.482,12.888,159.5253,0.0001,-2340.0000
C01315=-5.562,-97.322,12.887,159.5467,1.2343,-2343.2709
C01316=-10.602,-96.908,12.888,159.6590,2.1821,-2346.2435
C01317=-15.094,-96.401,12.910,160.4231,2.2511,-2348.8988
C01318=-18.135,-96.115,12.963,162.4714,0.9834,-2350.6850
C01319=-20.227,-96.057,13.031,165.7975,-0.3024,-2351.8912
C01320=-21.929,-96.117,13.096,169.6348,-0.5559,-2352.8520
C01321=-23.652,-96.157,13.142,173.0616,0.0823,-2353.8189
C01322=-25.795,-96.000,13.164,175.9036,0.5053,-2355.0400
C01323=-28.540,-95.542,13.175,178.1724,0.3760,-2356.6318
C01324=-31.535,-94.812,13.184,179.5717,0.1209,-2358.3974
C01325=-34.387,-93.888,13.193,179.9229,0.0278,-2360.1155
C01326=-37.002,-92.901,13.199,179.9912,0.0035,-2361.7171
C01327=-39.526,-91.855,13.199,179.9913,0.0038,-2363.2826
C01328=-42.074,-90.704,13.193,179.9258,0.0349,-2364.8847
C01329=-44.743,-89.341,13.184,179.6117,0.2174,-2366.6022
C01330=-47.377,-87.740,13.175,178.4418,1.0268,-2368.3677
C01331=-49.643,-86.123,13.164,176.7447,2.5426,-2369.9600
C01332=-51.269,-84.717,13.142,175.0240,4.8604,-2371.1815
C01333=-52.459,-83.471,13.096,173.0176,7.7557,-2372.1481
C01334=-53.620,-82.225,13.031,170.0612,10.3532,-2373.1089
C01335=-55.140,-80.787,12.963,166.7496,11.9257,-2374.3149
C01336=-57.492,-78.839,12.910,164.3969,12.6081,-2376.1008
C01337=-61.028,-76.021,12.888,163.8761,13.2352,-2378.7567
C01338=-64.884,-72.750,12.887,164.4132,13.9544,-2381.7290
C01339=-68.930,-68.930,12.888,165.2103,14.7899,-2385.0000
C01340=-72.750,-64.884,12.887,166.0456,15.5867,-2388.2710
C01341=-76.021,-61.028,12.888,166.7646,16.1238,-2391.2433
C01342=-78.839,-57.492,12.910,167.3920,15.6031,-2393.8992
C01343=-80.787,-55.140,12.963,168.0743,13.2504,-2395.6851
C01344=-82.225,-53.620,13.031,169.6468,9.9388,-2396.8911
C01345=-83.471,-52.459,13.096,172.2443,6.9824,-2397.8519
C01346=-84.717,-51.269,13.142,175.1396,4.9760,-2398.8185
C01347=-86.123,-49.643,13.164,177.4574,3.2553,-2400.0400
C01348=-87.740,-47.377,13.175,178.9732,1.5582,-2401.6323
C01349=-89.341,-44.743,13.184,179.7826,0.3883,-2403.3978
C01350=-90.704,-42.074,13.193,179.9651,0.0742,-2405.1153
C01351=-91.855,-39.526,13.199,179.9962,0.0087,-2406.7174
C01352=-92.901,-37.002,13.199,179.9965,0.0088,-2408.2829
C01353=-93.888,-34.387,13.193,179.9722,0.0771,-2409.8845
C01354=-94.812,-31.535,13.184,179.8791,0.4283,-2411.6026
C01355=-95.542,-28.540,13.175,179.6240,1.8276,-2413.3682
C01356=-96.000,-25.795,13.164,179.4947,4.0964,-2414.9600
C01357=-96.157,-23.652,13.142,179.9177,6.9384,-2416.1811
C01358=-96.117,-21.929,13.096,-179.4441,10.3652,-2417.1480
C01359=-96.057,-20.227,13.031,-179.6976,14.2025,-2418.1088
C01360=-96.115,-18.135,12.963,179.0166,17.5286,-2419.3150
C01361=-96.401,-15.094,12.910,177.7490,19.5770,-2421.1012
C01362=-96.908,-10.602,12.888,177.8177,20.3410,-2423.7565
C01363=-97.322,-5.562,12.887,178.7655,20.4533,-2426.7291
C01364=-97.482,0.000,12.888,-179.9999,20.4747,-2430.0000
C01365=-97.322,5.562,12.887,-178.7657,20.4533,-2433.2709
C01366=-96.908,10.602,12.888,-177.8179,20.3410,-2436.2435
C01367=-96.401,15.094,12.910,-177.7489,19.5769,-2438.8988
C01368=-96.115,18.135,12.963,-179.0166,17.5286,-2440.6850
C01369=-96.057,20.227,13.031,179.6976,14.2025,-2441.8912
C01370=-96.117,21.929,13.096,179.4441,10.3652,-2442.8520
C01371=-96.157,23.652,13.142,-179.9177,6.9384,-2443.8189
C01372=-96.000,25.795,13.164,-179.4947,4.0964,-2445.0400
C01373=-95.542,28.540,13.175,-179.6240,1.8276,-2446.6318
C01374=-94.812,31.535,13.184,-179.8791,0.4283,-2448.3974
C01375=-93.888,34.387,13.193,-179.9722,0.0771,-2450.1155
C01376=-92.901,37.002,13.199,-179.9965,0.0088,-2451.7171
C01377=-91.855,39.526,13.199,-179.9962,0.0087,-2453.2826
C01378=-90.704,42.074,13.193,-179.9651,0.0742,-2454.8847
C01379=-89.341,44.743,13.184,-179.7826,0.3883,-2456.6022
C01380=-87.740,47.377,13.175,-178.9732,1.5582,-2458.3677
C01381=-86.123,49.643,13.164,-177.4574,3.2553,-2459.9600
C01382=-84.717,51.269,13.142,-175.1396,4.9760,-2461.1815
C01383=-83.471,52.459,13.096,-172.2443,6.9824,-2462.1481
C01384=-82.225,53.620,13.031,-169.6468,9.9388,-2463.1089
C01385=-80.787,55.140,12.963,-168.0743,13.2504,-2464.3149
C01386=-78.839,57.492,12.910,-167.3919,15.6031,-2466.1008
C01387=-76.021,61.028,12.888,-166.7648,16.1239,-2468.7567
C01388=-72.750,64.884,12.887,-166.0456,15.5868,-2471.7290
C01389=-68.930,68.930,12.888,-165.2101,14.7897,-2475.0000
C01390=-64.884,72.750,12.887,-164.4133,13.9544,-2478.2710
C01391=-61.028,76.021,12.888,-163.8762,13.2354,-2481.2433
C01392=-57.492,78.839,12.910,-164.3969,12.6080,-2483.8992
C01393=-55.140,80.787,12.963,-166.7496,11.9257,-2485.6851
C01394=-53.620,82.225,13.031,-170.0612,10.3532,-2486.8911
C01395=-52.459,83.471,13.096,-173.0176,7.7557,-2487.8519
C01396=-51.269,84.717,13.142,-175.0240,4.8604,-2488.8185
C01397=-49.643,86.123,13.164,-176.7447,2.5426,-2490.0400
C01398=-47.377,87.740,13.175,-178.4418,1.0268,-2491.6323
C01399=-44.743,89.341,13.184,-179.6117,0.2174,-2493.3978
C01400=-42.074,90.704,13.193,-179.9258,0.0349,-2495.1153
C01401=-39.526,91.855,13.199,-179.9913,0.0038,-2496.7174
C01402=-37.002,92.901,13.199,-179.9912,0.0035,-2498.2829
C01403=-34.387,93.888,13.193,-179.9229,0.0278,-2499.8845
C01404=-31.535,94.812,13.184,-179.5717,0.1209,-2501.6026
C01405=-28.540,95.542,13.175,-178.1724,0.3760,-2503.3682
C01406=-25.795,96.000,13.164,-175.9036,0.5053,-2504.9600
C01407=-23.652,96.157,13.142,-173.0616,0.0823,-2506.1811
C01408=-21.929,96.117,13.096,-169.6348,-0.5559,-2507.1480
C01409=-20.227,96.057,13.031,-165.7975,-0.3024,-2508.1088
C01410=-18.135,96.115,12.963,-162.4714,0.9834,-2509.3150
C01411=-15.094,96.401,12.910,-160.4231,2.2511,-2511.1012
C01412=-10.602,96.908,12.888,-159.6590,2.1821,-2513.7565
C01413=-5.562,97.322,12.887,-159.5467,1.2343,-2516.7291
C01414=0.000,97.482,12.888,-159.5253,0.0001,-2520.0000
C01415=0.000,96.668,14.931,-157.0799,0.0002,-2520.0000
C01416=5.488,96.511,14.930,-157.1034,-1.3945,-2523.2546
C01417=10.476,96.104,14.932,-157.2237,-2.4088,-2526.2211
C01418=14.942,95.628,14.964,-158.0572,-2.1867,-2528.8807
C01419=17.951,95.422,15.043,-160.4780,-0.1533,-2530.6541
C01420=20.020,95.481,15.144,-164.5717,1.5921,-2531.8420
C01421=21.708,95.685,15.242,-169.0703,1.6612,-2532.7823
C01422=23.417,95.878,15.312,-172.7054,0.5194,-2533.7251
C01423=25.541,95.862,15.345,-175.6685,-0.3095,-2534.9190
C01424=28.302,95.513,15.362,-178.1073,-0.3286,-2536.5054
C01425=31.347,94.846,15.376,-179.5951,-0.1072,-2538.2889
C01426=34.268,93.927,15.390,-179.9213,-0.0281,-2540.0438
C01427=36.962,92.916,15.399,-179.9911,-0.0035,-2541.6927
C01428=39.566,91.838,15.399,-179.9913,-0.0038,-2543.3075
C01429=42.186,90.648,15.390,-179.9245,-0.0358,-2544.9564
C01430=44.901,89.232,15.376,-179.6379,-0.2105,-2546.7113
C01431=47.525,87.551,15.362,-178.4292,-1.1064,-2548.4943
C01432=49.724,85.845,15.345,-176.7161,-2.8475,-2550.0807
C01433=51.237,84.354,15.312,-175.1925,-5.5361,-2551.2747
C01434=52.309,83.010,15.242,-173.3810,-8.9256,-2552.2172
C01435=53.359,81.672,15.144,-170.0464,-12.1229,-2553.1579
C01436=54.780,80.167,15.043,-165.8238,-13.9722,-2554.3457
C01437=57.054,78.185,14.964,-162.6789,-14.4598,-2556.1194
C01438=60.548,75.364,14.932,-161.9108,-14.9574,-2558.7787
C01439=64.363,72.124,14.930,-162.4709,-15.7183,-2561.7455
C01440=68.355,68.355,14.931,-163.3542,-16.6460,-2565.0000
C01441=72.124,64.363,14.930,-164.2816,-17.5289,-2568.2545
C01442=75.364,60.548,14.932,-165.0425,-18.0890,-2571.2213
C01443=78.185,57.054,14.964,-165.5404,-17.3211,-2573.8806
C01444=80.167,54.780,15.043,-166.0278,-14.1762,-2575.6543
C01445=81.672,53.359,15.144,-167.8771,-9.9536,-2576.8421
C01446=83.010,52.309,15.242,-171.0744,-6.6190,-2577.7828
C01447=84.354,51.237,15.312,-174.4639,-4.8075,-2578.7253
C01448=85.845,49.724,15.345,-177.1525,-3.2839,-2579.9193
C01449=87.551,47.525,15.362,-178.8936,-1.5708,-2581.5057
C01450=89.232,44.901,15.376,-179.7895,-0.3621,-2583.2887
C01451=90.648,42.186,15.390,-179.9642,-0.0755,-2585.0436
C01452=91.838,39.566,15.399,-179.9962,-0.0087,-2586.6925
C01453=92.916,36.962,15.399,-179.9965,-0.0089,-2588.3073
C01454=93.927,34.268,15.390,-179.9719,-0.0787,-2589.9562
C01455=94.846,31.347,15.376,-179.8928,-0.4049,-2591.7111
C01456=95.513,28.302,15.362,-179.6714,-1.8927,-2593.4946
C01457=95.862,25.541,15.345,-179.6905,-4.3315,-2595.0810
C01458=95.878,23.417,15.312,179.4806,-7.2946,-2596.2749
C01459=95.685,21.708,15.242,178.3388,-10.9297,-2597.2177
C01460=95.481,20.020,15.144,178.4079,-15.4283,-2598.1580
C01461=95.422,17.951,15.043,-179.8467,-19.5220,-2599.3459
C01462=95.628,14.942,14.964,-177.8133,-21.9428,-2601.1193
C01463=96.104,10.476,14.932,-177.5912,-22.7763,-2603.7789
C01464=96.511,5.488,14.930,-178.6055,-22.8966,-2606.7454
C01465=96.668,0.000,14.931,179.9998,-22.9201,-2610.0000
C01466=96.511,-5.488,14.930,178.6057,-22.8966,-2613.2546
C01467=96.104,-10.476,14.932,177.5915,-22.7763,-2616.2211
C01468=95.628,-14.942,14.964,177.8131,-21.9428,-2618.8807
C01469=95.422,-17.951,15.043,179.8467,-19.5220,-2620.6541
C01470=95.481,-20.020,15.144,-178.4079,-15.4283,-2621.8420
C01471=95.685,-21.708,15.242,-178.3388,-10.9297,-2622.7823
C01472=95.878,-23.417,15.312,-179.4806,-7.2946,-2623.7251
C01473=95.862,-25.541,15.345,179.6905,-4.3315,-2624.9190
C01474=95.513,-28.302,15.362,179.6714,-1.8927,-2626.5054
C01475=94.846,-31.347,15.376,179.8928,-0.4049,-2628.2889
C01476=93.927,-34.268,15.390,179.9719,-0.0787,-2630.0438
C01477=92.916,-36.962,15.399,179.9965,-0.0089,-2631.6927
C01478=91.838,-39.566,15.399,179.9962,-0.0087,-2633.3075
C01479=90.648,-42.186,15.390,179.9642,-0.0755,-2634.9564
C01480=89.232,-44.901,15.376,179.7895,-0.3621,-2636.7113
C01481=87.551,-47.525,15.362,178.8936,-1.5708,-2638.4943
C01482=85.845,-49.724,15.345,177.1525,-3.2839,-2640.0807
C01483=84.354,-51.237,15.312,174.4639,-4.8075,-2641.2747
C01484=83.010,-52.309,15.242,171.0744,-6.6190,-2642.2172
C01485=81.672,-53.359,15.144,167.8771,-9.9536,-2643.1579
C01486=80.167,-54.780,15.043,166.0278,-14.1762,-2644.3457
C01487=78.185,-57.054,14.964,165.5402,-17.3211,-2646.1194
C01488=75.364,-60.548,14.932,165.0426,-18.0892,-2648.7787
C01489=72.124,-64.363,14.930,164.2817,-17.5291,-2651.7455
C01490=68.355,-68.355,14.931,163.3540,-16.6458,-2655.0000
C01491=64.363,-72.124,14.930,162.4711,-15.7184,-2658.2545
C01492=60.548,-75.364,14.932,161.9110,-14.9575,-2661.2213
C01493=57.054,-78.185,14.964,162.6789,-14.4596,-2663.8806
C01494=54.780,-80.167,15.043,165.8238,-13.9722,-2665.6543
C01495=53.359,-81.672,15.144,170.0464,-12.1229,-2666.8421
C01496=52.309,-83.010,15.242,173.3810,-8.9256,-2667.7828
C01497=51.237,-84.354,15.312,175.1925,-5.5361,-2668.7253
C01498=49.724,-85.845,15.345,176.7161,-2.8475,-2669.9193
C01499=47.525,-87.551,15.362,178.4292,-1.1064,-2671.5057
C01500=44.901,-89.232,15.376,179.6379,-0.2105,-2673.2887
C01501=42.186,-90.648,15.390,179.9245,-0.0358,-2675.0436
C01502=39.566,-91.838,15.399,179.9913,-0.0038,-2676.6925
C01503=36.962,-92.916,15.399,179.9911,-0.0035,-2678.3073
C01504=34.268,-93.927,15.390,179.9213,-0.0281,-2679.9562
C01505=31.347,-94.846,15.376,179.5951,-0.1072,-2681.7111
C01506=28.302,-95.513,15.362,178.1073,-0.3286,-2683.4946
C01507=25.541,-95.862,15.345,175.6685,-0.3095,-2685.0810
C01508=23.417,-95.878,15.312,172.7054,0.5194,-2686.2749
C01509=21.708,-95.685,15.242,169.0703,1.6612,-2687.2177
C01510=20.020,-95.481,15.144,164.5717,1.5921,-2688.1580
C01511=17.951,-95.422,15.043,160.4780,-0.1533,-2689.3459
C01512=14.942,-95.628,14.964,158.0572,-2.1867,-2691.1193
C01513=10.476,-96.104,14.932,157.2237,-2.4088,-2693.7789
C01514=5.488,-96.511,14.930,157.1034,-1.3945,-2696.7454
C01515=0.000,-96.668,14.931,157.0799,0.0002,-2700.0000
C01516=0.000,-96.668,14.931,157.0799,0.0002,-2700.0000
C01517=-5.488,-96.511,14.930,157.1034,1.3943,-2703.2546
C01518=-10.476,-96.104,14.932,157.2237,2.4085,-2706.2211
C01519=-14.942,-95.628,14.964,158.0572,2.1869,-2708.8807
C01520=-17.951,-95.422,15.043,160.4780,0.1533,-2710.6541
C01521=-20.020,-95.481,15.144,164.5717,-1.5921,-2711.8420
C01522=-21.708,-95.685,15.242,169.0703,-1.6612,-2712.7823
C01523=-23.417,-95.878,15.312,172.7054,-0.5194,-2713.7251
C01524=-25.541,-95.862,15.345,175.6685,0.3095,-2714.9190
C01525=-28.302,-95.513,15.362,178.1073,0.3286,-2716.5054
C01526=-31.347,-94.846,15.376,179.5951,0.1072,-2718.2889
C01527=-34.268,-93.927,15.390,179.9213,0.0281,-2720.0438
C01528=-36.962,-92.916,15.399,179.9911,0.0035,-2721.6927
C01529=-39.566,-91.838,15.399,179.9913,0.0038,-2723.3075
C01530=-42.186,-90.648,15.390,179.9245,0.0358,-2724.9564
C01531=-44.901,-89.232,15.376,179.6379,0.2105,-2726.7113
C01532=-47.525,-87.551,15.362,178.4292,1.1064,-2728.4943
C01533=-49.724,-85.845,15.345,176.7161,2.8475,-2730.0807
C01534=-51.237,-84.354,15.312,175.1925,5.5361,-2731.2747
C01535=-52.309,-83.010,15.242,173.3810,8.9256,-2732.2172
C01536=-53.359,-81.672,15.144,170.0464,12.1229,-2733.1579
C01537=-54.780,-80.167,15.043,165.8238,13.9722,-2734.3457
C01538=-57.054,-78.185,14.964,162.6789,14.4598,-2736.1194
C01539=-60.548,-75.364,14.932,161.9108,14.9574,-2738.7787
C01540=-64.363,-72.124,14.930,162.4709,15.7183,-2741.7455
C01541=-68.355,-68.355,14.931,163.3542,16.6460,-2745.0000
C01542=-72.124,-64.363,14.930,164.2816,17.5289,-2748.2545
C01543=-75.364,-60.548,14.932,165.0425,18.0890,-2751.2213
C01544=-78.185,-57.054,14.964,165.5404,17.3211,-2753.8806
C01545=-80.167,-54.780,15.043,166.0278,14.1762,-2755.6543
C01546=-81.672,-53.359,15.144,167.8771,9.9536,-2756.8421
C01547=-83.010,-52.309,15.242,171.0744,6.6190,-2757.7828
C01548=-84.354,-51.237,15.312,174.4639,4.8075,-2758.7253
C01549=-85.845,-49.724,15.345,177.1525,3.2839,-2759.9193
C01550=-87.551,-47.525,15.362,178.8936,1.5708,-2761.5057
C01551=-89.232,-44.901,15.376,179.7895,0.3621,-2763.2887
C01552=-90.648,-42.186,15.390,179.9642,0.0755,-2765.0436
C01553=-91.838,-39.566,15.399,179.9962,0.0087,-2766.6925
C01554=-92.916,-36.962,15.399,179.9965,0.0089,-2768.3073
C01555=-93.927,-34.268,15.390,179.9719,0.0787,-2769.9562
C01556=-94.846,-31.347,15.376,179.8928,0.4049,-2771.7111
C01557=-95.513,-28.302,15.362,179.6714,1.8927,-2773.4946
C01558=-95.862,-25.541,15.345,179.6905,4.3315,-2775.0810
C01559=-95.878,-23.417,15.312,-179.4806,7.2946,-2776.2749
C01560=-95.685,-21.708,15.242,-178.3388,10.9297,-2777.2177
C01561=-95.481,-20.020,15.144,-178.4079,15.4283,-2778.1580
C01562=-95.422,-17.951,15.043,179.8467,19.5220,-2779.3459
C01563=-95.628,-14.942,14.964,177.8133,21.9428,-2781.1193
C01564=-96.104,-10.476,14.932,177.5912,22.7763,-2783.7789
C01565=-96.511,-5.488,14.930,178.6055,22.8966,-2786.7454
C01566=-96.668,0.000,14.931,-179.9998,22.9201,-2790.0000
C01567=-96.511,5.488,14.930,-178.6057,22.8966,-2793.2546
C01568=-96.104,10.476,14.932,-177.5915,22.7763,-2796.2211
C01569=-95.628,14.942,14.964,-177.8131,21.9428,-2798.8807
C01570=-95.422,17.951,15.043,-179.8467,19.5220,-2800.6541
C01571=-95.481,20.020,15.144,178.4079,15.4283,-2801.8420
C01572=-95.685,21.708,15.242,178.3388,10.9297,-2802.7823
C01573=-95.878,23.417,15.312,179.4806,7.2946,-2803.7251
C01574=-95.862,25.541,15.345,-179.6905,4.3315,-2804.9190
C01575=-95.513,28.302,15.362,-179.6714,1.8927,-2806.5054
C01576=-94.846,31.347,15.376,-179.8928,0.4049,-2808.2889
C01577=-93.927,34.268,15.390,-179.9719,0.0787,-2810.0438
C01578=-92.916,36.962,15.399,-179.9965,0.0089,-2811.6927
C01579=-91.838,39.566,15.399,-179.9962,0.0087,-2813.3075
C01580=-90.648,42.186,15.390,-179.9642,0.0755,-2814.9564
C01581=-89.232,44.901,15.376,-179.7895,0.3621,-2816.7113
C01582=-87.551,47.525,15.362,-178.8936,1.5708,-2818.4943
C01583=-85.845,49.724,15.345,-177.1525,3.2839,-2820.0807
C01584=-84.354,51.237,15.312,-174.4639,4.8075,-2821.2747
C01585=-83.010,52.309,15.242,-171.0744,6.6190,-2822.2172
C01586=-81.672,53.359,15.144,-167.8771,9.9536,-2823.1579
C01587=-80.167,54.780,15.043,-166.0278,14.1762,-2824.3457
C01588=-78.185,57.054,14.964,-165.5402,17.3211,-2826.1194
C01589=-75.364,60.548,14.932,-165.0426,18.0892,-2828.7787
C01590=-72.124,64.363,14.930,-164.2817,17.5291,-2831.7455
C01591=-68.355,68.355,14.931,-163.3540,16.6458,-2835.0000
C01592=-64.363,72.124,14.930,-162.4711,15.7184,-2838.2545
C01593=-60.548,75.364,14.932,-161.9110,14.9575,-2841.2213
C01594=-57.054,78.185,14.964,-162.6789,14.4596,-2843.8806
C01595=-54.780,80.167,15.043,-165.8238,13.9722,-2845.6543
C01596=-53.359,81.672,15.144,-170.0464,12.1229,-2846.8421
C01597=-52.309,83.010,15.242,-173.3810,8.9256,-2847.7828
C01598=-51.237,84.354,15.312,-175.1925,5.5361,-2848.7253
C01599=-49.724,85.845,15.345,-176.7161,2.8475,-2849.9193
C01600=-47.525,87.551,15.362,-178.4292,1.1064,-2851.5057
C01601=-44.901,89.232,15.376,-179.6379,0.2105,-2853.2887
C01602=-42.186,90.648,15.390,-179.9245,0.0358,-2855.0436
C01603=-39.566,91.838,15.399,-179.9913,0.0038,-2856.6925
C01604=-36.962,92.916,15.399,-179.9911,0.0035,-2858.3073
C01605=-34.268,93.927,15.390,-179.9213,0.0281,-2859.9562
C01606=-31.347,94.846,15.376,-179.5951,0.1072,-2861.7111
C01607=-28.302,95.513,15.362,-178.1073,0.3286,-2863.4946
C01608=-25.541,95.862,15.345,-175.6685,0.3095,-2865.0810
C01609=-23.417,95.878,15.312,-172.7054,-0.5194,-2866.2749
C01610=-21.708,95.685,15.242,-169.0703,-1.6612,-2867.2177
C01611=-20.020,95.481,15.144,-164.5717,-1.5921,-2868.1580
C01612=-17.951,95.422,15.043,-160.4780,0.1533,-2869.3459
C01613=-14.942,95.628,14.964,-158.0572,2.1869,-2871.1193
C01614=-10.476,96.104,14.932,-157.2237,2.4085,-2873.7789
C01615=-5.488,96.511,14.930,-157.1034,1.3943,-2876.7454
C01616=0.000,96.668,14.931,-157.0799,0.0002,-2880.0000
C01617=0.000,95.772,16.941,-154.8859,0.0002,-2880.0000
C01618=5.406,95.617,16.939,-154.9111,-1.5415,-2883.2359
C01619=10.339,95.219,16.941,-155.0372,-2.5925,-2886.1970
C01620=14.774,94.777,16.986,-155.9394,-1.9734,-2888.8601
C01621=17.748,94.656,17.095,-158.8449,1.0095,-2890.6197
C01622=19.790,94.842,17.237,-163.9074,3.1515,-2891.7864
C01623=21.462,95.203,17.374,-169.0788,2.8690,-2892.7041
C01624=23.155,95.565,17.473,-172.7347,1.2030,-2893.6200
C01625=25.257,95.708,17.521,-175.6219,-0.0566,-2894.7831
C01626=28.035,95.481,17.545,-178.1277,-0.2593,-2896.3632
C01627=31.135,94.884,17.565,-179.6493,-0.0862,-2898.1666
C01628=34.135,93.972,17.585,-179.9232,-0.0272,-2899.9634
C01629=36.917,92.934,17.598,-179.9915,-0.0033,-2901.6649
C01630=39.610,91.818,17.598,-179.9916,-0.0037,-2903.3352
C01631=42.311,90.585,17.585,-179.9265,-0.0351,-2905.0366
C01632=45.077,89.109,17.565,-179.6910,-0.1870,-2906.8332
C01633=47.692,87.339,17.545,-178.4926,-1.1409,-2908.6370
C01634=49.816,85.535,17.521,-176.8613,-3.0589,-2910.2167
C01635=51.202,83.948,17.473,-175.6939,-5.9938,-2911.3801
C01636=52.143,82.495,17.374,-174.2326,-9.7525,-2912.2959
C01637=53.070,81.058,17.237,-170.6271,-13.6544,-2913.2134
C01638=54.382,79.482,17.095,-165.3630,-15.9654,-2914.3801
C01639=56.571,77.464,16.986,-161.2176,-16.2439,-2916.1402
C01640=60.019,74.640,16.941,-160.1409,-16.5495,-2918.8032
C01641=63.789,71.434,16.939,-160.7051,-17.3299,-2921.7642
C01642=67.721,67.721,16.941,-161.6626,-18.3377,-2925.0000
C01643=71.434,63.789,16.939,-162.6700,-19.2947,-2928.2358
C01644=74.640,60.019,16.941,-163.4503,-19.8589,-2931.1968
C01645=77.464,56.571,16.986,-163.7563,-18.7825,-2933.8598
C01646=79.482,54.382,17.095,-164.0346,-14.6370,-2935.6199
C01647=81.058,53.070,17.237,-166.3456,-9.3729,-2936.7866
C01648=82.495,52.143,17.374,-170.2475,-5.7674,-2937.7041
C01649=83.948,51.202,17.473,-174.0062,-4.3061,-2938.6199
C01650=85.535,49.816,17.521,-176.9411,-3.1387,-2939.7833
C01651=87.339,47.692,17.545,-178.8591,-1.5074,-2941.3630
C01652=89.109,45.077,17.565,-179.8130,-0.3090,-2943.1668
C01653=90.585,42.311,17.585,-179.9649,-0.0735,-2944.9634
C01654=91.818,39.610,17.598,-179.9963,-0.0084,-2946.6648
C01655=92.934,36.917,17.598,-179.9967,-0.0085,-2948.3351
C01656=93.972,34.135,17.585,-179.9728,-0.0768,-2950.0366
C01657=94.884,31.135,17.565,-179.9138,-0.3507,-2951.8334
C01658=95.481,28.035,17.545,-179.7407,-1.8723,-2953.6368
C01659=95.708,25.257,17.521,-179.9434,-4.3781,-2955.2169
C01660=95.565,23.155,17.473,178.7970,-7.2653,-2956.3800
C01661=95.203,21.462,17.374,177.1310,-10.9212,-2957.2959
C01662=94.842,19.790,17.237,176.8485,-16.0926,-2958.2136
C01663=94.656,17.748,17.095,178.9905,-21.1551,-2959.3803
C01664=94.777,14.774,16.986,-178.0266,-24.0606,-2961.1399
C01665=95.219,10.339,16.941,-177.4075,-24.9628,-2963.8030
C01666=95.617,5.406,16.939,-178.4585,-25.0889,-2966.7641
C01667=95.772,0.000,16.941,179.9998,-25.1141,-2970.0000
C01668=95.617,-5.406,16.939,178.4588,-25.0889,-2973.2359
C01669=95.219,-10.339,16.941,177.4079,-24.9628,-2976.1970
C01670=94.777,-14.774,16.986,178.0264,-24.0606,-2978.8601
C01671=94.656,-17.748,17.095,-178.9905,-21.1551,-2980.6197
C01672=94.842,-19.790,17.237,-176.8485,-16.0926,-2981.7864
C01673=95.203,-21.462,17.374,-177.1310,-10.9212,-2982.7041
C01674=95.565,-23.155,17.473,-178.7970,-7.2653,-2983.6200
C01675=95.708,-25.257,17.521,179.9434,-4.3781,-2984.7831
C01676=95.481,-28.035,17.545,179.7407,-1.8723,-2986.3632
C01677=94.884,-31.135,17.565,179.9138,-0.3507,-2988.1666
C01678=93.972,-34.135,17.585,179.9728,-0.0768,-2989.9634
C01679=92.934,-36.917,17.598,179.9967,-0.0085,-2991.6649
C01680=91.818,-39.610,17.598,179.9963,-0.0084,-2993.3352
C01681=90.585,-42.311,17.585,179.9649,-0.0735,-2995.0366
C01682=89.109,-45.077,17.565,179.8130,-0.3090,-2996.8332
C01683=87.339,-47.692,17.545,178.8591,-1.5074,-2998.6370
C01684=85.535,-49.816,17.521,176.9411,-3.1387,-3000.2167
C01685=83.948,-51.202,17.473,174.0062,-4.3061,-3001.3801
C01686=82.495,-52.143,17.374,170.2475,-5.7674,-3002.2959
C01687=81.058,-53.070,17.237,166.3456,-9.3729,-3003.2134
C01688=79.482,-54.382,17.095,164.0346,-14.6370,-3004.3801
C01689=77.464,-56.571,16.986,163.7561,-18.7824,-3006.1402
C01690=74.640,-60.019,16.941,163.4505,-19.8591,-3008.8032
C01691=71.434,-63.789,16.939,162.6701,-19.2949,-3011.7642
C01692=67.721,-67.721,16.941,161.6623,-18.3374,-3015.0000
C01693=63.789,-71.434,16.939,160.7053,-17.3300,-3018.2358
C01694=60.019,-74.640,16.941,160.1411,-16.5497,-3021.1968
C01695=56.571,-77.464,16.986,161.2175,-16.2437,-3023.8598
C01696=54.382,-79.482,17.095,165.3630,-15.9654,-3025.6199
C01697=53.070,-81.058,17.237,170.6271,-13.6544,-3026.7866
C01698=52.143,-82.495,17.374,174.2326,-9.7525,-3027.7041
C01699=51.202,-83.948,17.473,175.6939,-5.9938,-3028.6199
C01700=49.816,-85.535,17.521,176.8613,-3.0589,-3029.7833
C01701=47.692,-87.339,17.545,178.4926,-1.1409,-3031.3630
C01702=45.077,-89.109,17.565,179.6910,-0.1870,-3033.1668
C01703=42.311,-90.585,17.585,179.9265,-0.0351,-3034.9634
C01704=39.610,-91.818,17.598,179.9916,-0.0037,-3036.6648
C01705=36.917,-92.934,17.598,179.9915,-0.0033,-3038.3351
C01706=34.135,-93.972,17.585,179.9232,-0.0272,-3040.0366
C01707=31.135,-94.884,17.565,179.6493,-0.0862,-3041.8334
C01708=28.035,-95.481,17.545,178.1277,-0.2593,-3043.6368
C01709=25.257,-95.708,17.521,175.6219,-0.0566,-3045.2169
C01710=23.155,-95.565,17.473,172.7347,1.2030,-3046.3800
C01711=21.462,-95.203,17.374,169.0788,2.8690,-3047.2959
C01712=19.790,-94.842,17.237,163.9074,3.1515,-3048.2136
C01713=17.748,-94.656,17.095,158.8449,1.0095,-3049.3803
C01714=14.774,-94.777,16.986,155.9394,-1.9734,-3051.1399
C01715=10.339,-95.219,16.941,155.0372,-2.5925,-3053.8030
C01716=5.406,-95.617,16.939,154.9111,-1.5415,-3056.7641
C01717=0.000,-95.772,16.941,154.8859,0.0002,-3060.0000
C01718=0.000,-95.772,16.941,154.8859,0.0002,-3060.0000
C01719=-5.406,-95.617,16.939,154.9111,1.5412,-3063.2359
C01720=-10.339,-95.219,16.941,155.0372,2.5921,-3066.1970
C01721=-14.774,-94.777,16.986,155.9394,1.9736,-3068.8601
C01722=-17.748,-94.656,17.095,158.8449,-1.0095,-3070.6197
C01723=-19.790,-94.842,17.237,163.9074,-3.1515,-3071.7864
C01724=-21.462,-95.203,17.374,169.0788,-2.8690,-3072.7041
C01725=-23.155,-95.565,17.473,172.7347,-1.2030,-3073.6200
C01726=-25.257,-95.708,17.521,175.6219,0.0566,-3074.7831
C01727=-28.035,-95.481,17.545,178.1277,0.2593,-3076.3632
C01728=-31.135,-94.884,17.565,179.6493,0.0862,-3078.1666
C01729=-34.135,-93.972,17.585,179.9232,0.0272,-3079.9634
C01730=-36.917,-92.934,17.598,179.9915,0.0033,-3081.6649
C01731=-39.610,-91.818,17.598,179.9916,0.0037,-3083.3352
C01732=-42.311,-90.585,17.585,179.9265,0.0351,-3085.0366
C01733=-45.077,-89.109,17.565,179.6910,0.1870,-3086.8332
C01734=-47.692,-87.339,17.545,178.4926,1.1409,-3088.6370
C01735=-49.816,-85.535,17.521,176.8613,3.0589,-3090.2167
C01736=-51.202,-83.948,17.473,175.6939,5.9938,-3091.3801
C01737=-52.143,-82.495,17.374,174.2326,9.7525,-3092.2959
C01738=-53.070,-81.058,17.237,170.6271,13.6544,-3093.2134
C01739=-54.382,-79.482,17.095,165.3630,15.9654,-3094.3801
C01740=-56.571,-77.464,16.986,161.2176,16.2439,-3096.1402
C01741=-60.019,-74.640,16.941,160.1409,16.5495,-3098.8032
C01742=-63.789,-71.434,16.939,160.7051,17.3299,-3101.7642
C01743=-67.721,-67.721,16.941,161.6626,18.3377,-3105.0000
C01744=-71.434,-63.789,16.939,162.6700,19.2947,-3108.2358
C01745=-74.640,-60.019,16.941,163.4503,19.8589,-3111.1968
C01746=-77.464,-56.571,16.986,163.7563,18.7825,-3113.8598
C01747=-79.482,-54.382,17.095,164.0346,14.6370,-3115.6199
C01748=-81.058,-53.070,17.237,166.3456,9.3729,-3116.7866
C01749=-82.495,-52.143,17.374,170.2475,5.7674,-3117.7041
C01750=-83.948,-51.202,17.473,174.0062,4.3061,-3118.6199
C01751=-85.535,-49.816,17.521,176.9411,3.1387,-3119.7833
C01752=-87.339,-47.692,17.545,178.8591,1.5074,-3121.3630
C01753=-89.109,-45.077,17.565,179.8130,0.3090,-3123.1668
C01754=-90.585,-42.311,17.585,179.9649,0.0735,-3124.9634
C01755=-91.818,-39.610,17.598,179.9963,0.0084,-3126.6648
C01756=-92.934,-36.917,17.598,179.9967,0.0085,-3128.3351
C01757=-93.972,-34.135,17.585,179.9728,0.0768,-3130.0366
C01758=-94.884,-31.135,17.565,179.9138,0.3507,-3131.8334
C01759=-95.481,-28.035,17.545,179.7407,1.8723,-3133.6368
C01760=-95.708,-25.257,17.521,179.9434,4.3781,-3135.2169
C01761=-95.565,-23.155,17.473,-178.7970,7.2653,-3136.3800
C01762=-95.203,-21.462,17.374,-177.1310,10.9212,-3137.2959
C01763=-94.842,-19.790,17.237,-176.8485,16.0926,-3138.2136
C01764=-94.656,-17.748,17.095,-178.9905,21.1551,-3139.3803
C01765=-94.777,-14.774,16.986,178.0266,24.0606,-3141.1399
C01766=-95.219,-10.339,16.941,177.4075,24.9628,-3143.8030
C01767=-95.617,-5.406,16.939,178.4585,25.0889,-3146.7641
C01768=-95.772,0.000,16.941,-179.9998,25.1141,-3150.0000
C01769=-95.617,5.406,16.939,-178.4588,25.0889,-3153.2359
C01770=-95.219,10.339,16.941,-177.4079,24.9628,-3156.1970
C01771=-94.777,14.774,16.986,-178.0264,24.0606,-3158.8601
